(* Logix 5000 project; controller LeakTestAuto vendor 1 type 14 code 226 rev 37.11; software revision 37.01 *)

TASK MainTask (continuous, watchdog 500 ms) : MainProgram
TASK SafetyTask (periodic, rate 20 ms, priority 10, watchdog 20 ms, safety) : SafetyProgram

MODULES
   Local : vendor 1 type 14 code 226 (5069 0, rev 37.11)
      Main : vendor 1 type 14 code 195 (Ethernet 192.168.1.210, rev 33.1, $87205a54$ RPI 20 ms)
       : 5069-IB8S (5069 1, rev 2.1, SafetyInput RPI 20 ms)
      Barcode : vendor 367 type 43 code 1009 (Ethernet 192.168.1.214, rev 1.1, StandardDataDriven RPI 20 ms)
      CTS1 : vendor 1415 type 43 code 9245 (Ethernet 192.168.1.212, rev 1.1, StandardDataDriven RPI 25 ms)
      CTS2 : vendor 1415 type 43 code 9245 (Ethernet 192.168.1.213, rev 1.1, StandardDataDriven RPI 25 ms)
      EpsonRobot : vendor 1009 type 43 code 9 (Ethernet 192.168.1.215, rev 1.2, StandardDataDriven RPI 10 ms)
       : 5069-IB16 (5069 3, rev 2.1, StandardDataDriven RPI 5 ms)
       : 5069-OB16 (5069 5, rev 3.1, StandardDataDriven RPI 5 ms)
       : 5069-IB16 (5069 4, rev 2.1, StandardDataDriven RPI 5 ms)
       : 5069-OBV8S (5069 2, rev 1.1, SafetyInput RPI 20 ms)
      RFID : vendor 322 type 43 code 102 (Ethernet 192.168.1.217, rev 4.2, StandardDataDriven RPI 10 ms)
      DTE102_RFID_LoadingNest : vendor 322 type 43 code 102 (Ethernet 192.168.1.218, rev 4.2, StandardDataDriven RPI 10 ms)
END_MODULES

TYPE DTE102_CmdModule :   // It handles the imapping of the DTE102 command and status
STRUCT
   ActivateCommand : DTE102_OutputBits;   // Used to give commmands to DTE102 from PLC
   Status : DTE102_InputBits;   // Used to read the status from the DTE102 to PLC
END_STRUCT
END_TYPE

TYPE DTE102_InputBits :   // List of Bits used in PLC Input Image
STRUCT
   TP : BOOL;   // Byte 1, Bit 0 - Tag Present Status
   AI : BOOL;   // Byte 1, Bit 1 - Antenna Inactive Status
   WA : BOOL;   // Byte 1, bit 2 - Mode Write Data ACTIVE
   RA : BOOL;   // Byte 1, bit 3 - Mode Read Data ACTIVE
   UA : BOOL;   // Byte 1, bit 4 - Mode User Data Access ACTIVE
   EA : BOOL;   // Byte 1, bit 5 - Mode Receive User Data on Event Change ACTIVE
   DA : BOOL;   // Byte 1, bit 6 - Mode Diagnostics Read ACTIVE
   DIAG : BOOL;   // Byte 1, bit 7 - DIAGnostic Data Present
   TA : BOOL;   // Byte 2, bit 0 - Toggle Request Acknowledge
   CA : BOOL;   // Byte 2, bit 7 - Command Mode Active
END_STRUCT
END_TYPE

TYPE DTE102_OutputBits :   // List of Bits used in PLC Output Image
STRUCT
   AO : BOOL;   // Byte 1, Bit 1 - Antenna Inactive Request
   WR : BOOL;   // Byte 1, bit 2 - Mode Write Data ACTIVATE Command
   RD : BOOL;   // Byte 1, bit 3 - Mode Read Data ACTIVATE Command
   UR : BOOL;   // Byte 1, bit 4 - Mode User Data Access ACTIVATE Command
   ER : BOOL;   // Byte 1, bit 5 - Event Controlled reading of user memory of the ID tag
   DR : BOOL;   // Byte 1, bit 6 - Mode Diagnostics Read
   TR : BOOL;   // Byte 2, bit 0 - Toggle Request
   CM : BOOL;   // Byte 2, bit 7 - Command Mode Activate
END_STRUCT
END_TYPE

TYPE STR_Barcode :
STRUCT
   LEN : DINT;
   DATA : SINT[128];
END_STRUCT
END_TYPE

TYPE STRING16 :
STRUCT
   LEN : DINT;
   DATA : SINT[16];
END_STRUCT
END_TYPE

TYPE String20 :
STRUCT
   LEN : DINT;
   DATA : SINT[20];
END_STRUCT
END_TYPE

TYPE String35 :
STRUCT
   LEN : DINT;
   DATA : SINT[35];
END_STRUCT
END_TYPE

TYPE STRING80 :
STRUCT
   LEN : DINT;
   DATA : SINT[80];
END_STRUCT
END_TYPE

TYPE udt_CTS_INPUTS_FROM :
STRUCT
   Discrete_Status_Data : INT;   // Discrete Type Instrument Outputs
   Discrete_User_Output : INT;   // Control Commands
   Active_program_num : INT;   // Current program number
   Active_child_program : INT;   // required for alignment
   unique_id : DINT;   // Unique Identifier for the most recent result
   channel_num : SINT;   // Channel number for the most recent result
   Reserved_4 : SINT;
   Reserved_5 : SINT;
   Reserved_6 : SINT;
   program_num : INT;   // Program number for the most recent result
   sequence_num : INT;   // Test Port number for the most recent result
   seq_unique_ID : DINT;   // UID of seq program
   evaluation_code : INT;   // Evaluation code for the most recent result
   test_port : SINT;   // Test Port
   year : SINT;   // Timestamp year (YY) for the most recent result
   month : SINT;   // Timestamp month (MM) for the most recent result
   date : SINT;   // Timestamp day (DD) for the most recent result
   hour : SINT;   // Timestamp hour (HH) for the most recent result
   minutes : SINT;   // Timestamp minute (MM) for the most recent result
   seconds : SINT;   // Timestamp second (SS) for the most recent result
   flags : SINT;   // Result flags
   test_type : INT;   // Test Type
   Segment_code : INT;
   Measurement_data : udt_CTS_Measurement_Element[4];
END_STRUCT
END_TYPE

TYPE udt_CTS_Measurement_Element :
STRUCT
   Variable_code : INT;
   Variable_Number : SINT;
   Precision_code : SINT;
   Unit_code : INT;
   Reserved_1 : SINT;
   Reserved_2 : SINT;
   result_measurement : REAL;
END_STRUCT
END_TYPE

TYPE udt_CTS_OUTPUTS_TO :
STRUCT
   reserved : BOOL;   // reserved1
   change_program : BOOL;   // out_value 1
   Latch_2_Clear : BOOL;   // out_value 2
   Latch_2_Set : BOOL;   // out_value 3
   Latch_1_Clear : BOOL;   // out_value 4
   Latch_1_Set : BOOL;   // out_value 5
   New_Result_Clear : BOOL;   // out_value 6
   Requested_Result_Clear : BOOL;   // out_value 7
   reserved_2 : BOOL;   // out_value 8
   reserved_3 : BOOL;   // out_value 9
   reerved_4 : BOOL;   // out_value 10
   reserved_5 : BOOL;   // out_value 11
   vent_halt : BOOL;   // out_value 12
   reset : BOOL;   // out_value 13
   Stop : BOOL;   // out_value 14
   Start_channel : BOOL;   // out_value 15
   Out_val_1 : BOOL;   // out_value 16
   Out_val_2 : BOOL;   // Change_Program
   Out_val_3 : BOOL;   // Latch_2_Clear
   Out_val_4 : BOOL;   // Latch_2_Set
   Out_val_5 : BOOL;   // Latch_1_Clear
   Out_val_6 : BOOL;   // Latch_1_Set
   Out_val_7 : BOOL;   // New Result Clear
   Out_val_8 : BOOL;   // Requested Result Clear
   Out_val_9 : BOOL;   // reserved3
   Out_val_10 : BOOL;   // reserved4
   Out_val_11 : BOOL;   // reserved5
   Out_val_12 : BOOL;   // reserved6
   Out_val_13 : BOOL;   // VentHalt
   Out_val_14 : BOOL;   // Reset
   Out_val_15 : BOOL;   // Stop
   Out_val_16 : BOOL;   // Start_Channel
   program_num : INT;   // program_num
END_STRUCT
END_TYPE

TYPE udt_CTS_RESULT :
STRUCT
   UID : DINT;
   Basic : udt_CTS_RESULT_BASIC;
   Detailed : udt_CTS_RESULT_DETAILED;
END_STRUCT
END_TYPE

TYPE udt_CTS_RESULT_BASIC :
STRUCT
   unique_id : DINT;
   channel_num : SINT;
   reserved1 : SINT;
   reserved2 : SINT;
   reserved3 : SINT;
   program_num : INT;
   sequence_num : SINT;
   seq_unique_ID : DINT;
   evaluation_code : INT;
   test_port : SINT;
   year : SINT;
   month : SINT;
   date : SINT;
   hour : SINT;
   minute : SINT;
   second : SINT;
   reserved_4 : SINT;
   flags : SINT;
   reserved_5 : SINT;
   barcode_characters : SINT[80];
   Num_tests : SINT;
   reserved_6 : SINT;
   reserved_7 : SINT;
   reserved_8 : SINT;
   test_elements : udt_CTS_RESULT_BASIC_TEST_ELEMENT;
   barcode : STRING80;
END_STRUCT
END_TYPE

TYPE udt_CTS_RESULT_BASIC_TEST_ELEMENT :
STRUCT
   test_type : INT;
   test_eval : INT;
   num_elements : SINT;
   reserved1 : SINT;
END_STRUCT
END_TYPE

TYPE udt_CTS_RESULT_DETAILED :
STRUCT
   unique_id : DINT;
   num_elements : SINT;
   reserved_1 : SINT;
   Test_Type : INT;
   element_data : udt_CTS_RESULT_DETAILED_DATA_ELEMENT[30];
   reserved_2 : SINT;
   reserved_3 : SINT;
END_STRUCT
END_TYPE

TYPE udt_CTS_RESULT_DETAILED_DATA_ELEMENT :
STRUCT
   Variable_code : INT;
   variable_Num : SINT;
   prec_code : SINT;
   Unit_code : INT;
   reserved1 : SINT;
   reserved2 : SINT;
   result_measurement : REAL;
END_STRUCT
END_TYPE

TYPE udt_DUTHistory :
STRUCT
   Barcode : STR_Barcode;
   VolumeTest : REAL;
   LeakTest : REAL;
END_STRUCT
END_TYPE

TYPE udt_EIPTemplateData :
STRUCT
   Data : SINT[64];
END_STRUCT
END_TYPE

TYPE udt_EIPTemplateLocalInput :
STRUCT
   Ready : BOOL;
   Error : BOOL;
   Busy : BOOL;
   DataAvailable : BOOL;
   Complete : BOOL;
   Spare5 : BOOL;
   Spare6 : BOOL;
   Spare7 : BOOL;
   Data : SINT[8];
   SpareB9_63 : SINT[55];
END_STRUCT
END_TYPE

TYPE udt_EIPTemplateLocalOutput :
STRUCT
   Start : BOOL;
   Stop : BOOL;
   GetData : BOOL;
   Spare3 : BOOL;
   Spare4 : BOOL;
   Spare5 : BOOL;
   Spare6 : BOOL;
   Spare7 : BOOL;
   SpareB1_63 : SINT[63];
END_STRUCT
END_TYPE

TYPE udt_EpsonInputs :
STRUCT
   ib_Initializing : BOOL;
   ib_Ready : BOOL;
   ib_Running : BOOL;
   ib_Paused : BOOL;
   ib_Error : BOOL;
   ib_EStop : BOOL;
   ib_MotorsOn : BOOL;
   ib_IsHome : BOOL;
   ib_InPos : BOOL;
   ib_GripOpen : BOOL;
   ib_GripClosed : BOOL;
   SPAREB13 : BOOL;
   SPAREB14 : BOOL;
   SPAREB15 : BOOL;
   SPAREB16 : BOOL;
   SPAREB17 : BOOL;
   iB_SpeedEcho : USINT;
   SPAREB307 : USINT;
   iB_AccEcho : USINT;
   iB_DecEcho : USINT;
   SPAREW4 : UINT;
   SPAREW5 : UINT;
   SPAREW6 : UINT;
   SPAREW7 : UINT;
   iW_PositionEcho : UINT;
   iR_X : REAL;
   iR_Y : REAL;
   iR_Z : REAL;
   iR_U : REAL;
END_STRUCT
END_TYPE

TYPE udt_EpsonOutputs :
STRUCT
   ob_Start : BOOL;
   ob_StopNOTUSED : BOOL;
   ob_Resume : BOOL;
   ob_Pause : BOOL;
   ob_Reset : BOOL;
   ob_GoHome : BOOL;
   SPAREB06 : BOOL;
   SPAREB07 : BOOL;
   ob_SpeedOverride : BOOL;
   ob_AccOverride : BOOL;
   ob_CoordMode : BOOL;
   SPAREB13 : BOOL;
   SPAREB14 : BOOL;
   SPAREB15 : BOOL;
   SPAREB16 : BOOL;
   SPAREB17 : BOOL;
   oB_SpeedPerc : USINT;
   SPAREB307 : USINT;
   oB_AccPerc : USINT;
   oB_DecPerc : USINT;
   SPAREW4 : UINT;
   SPAREW5 : UINT;
   SPAREW6 : UINT;
   SPAREW7 : UINT;
   oW_TargetPosition : UINT;
   oR_X : REAL;
   oR_Y : REAL;
   oR_Z : REAL;
   oR_U : REAL;
END_STRUCT
END_TYPE

TYPE udt_KeyenceScannerInputs :
STRUCT
   Error : BOOL;
   ResultDataAvailable : BOOL;
   ResultDataStrobe : BOOL;
   Reserve0_3 : BOOL;
   Reserve0_4 : BOOL;
   Reserve0_5 : BOOL;
   BufferOverflowError : BOOL;
   GeneralError : BOOL;
   BUSY : BOOL;
   TRGBUSY : BOOL;
   LOCKBUSY : BOOL;
   MODEBUSY : BOOL;
   ERRBUSY : BOOL;
   Reserve0_13 : BOOL;
   READY : BOOL;
   Reserve0_15 : BOOL;
   ReadComplete : BOOL;
   PresetComplete : BOOL;
   RegisterPresetDataComplete : BOOL;
   TuneComplete : BOOL;
   BloadComplete : BOOL;
   Reserve2_5 : BOOL;
   Reserve2_6 : BOOL;
   EXTRequestComplete : BOOL;
   ReadFailure : BOOL;
   PresetFailure : BOOL;
   RegisterPresetDataFailure : BOOL;
   TuneFailure : BOOL;
   BloadFailure : BOOL;
   Reserve2_13 : BOOL;
   Reserve2_14 : BOOL;
   EXTRequestFailure : BOOL;
   IN1Status : BOOL;
   IN2Status : BOOL;
   Reserve4_2 : BOOL;
   Reserve4_3 : BOOL;
   OUT1Status : BOOL;
   OUT2Status : BOOL;
   OUT3Status : BOOL;
   Reserve4_7 : BOOL;
   Unstable : BOOL;
   MatchingLevelUnstable : BOOL;
   ISOIEC15415Unstable : BOOL;
   AIMDPMUnstable : BOOL;
   SAEAS9132Unstable : BOOL;
   ISOIEC15416Unstable : BOOL;
   Reserve4_14 : BOOL;
   Reserve4_15 : BOOL;
   Reserve6_0 : BOOL;
   Reserve6_1 : BOOL;
   Reserve6_2 : BOOL;
   Reserve6_3 : BOOL;
   Reserve6_4 : BOOL;
   Reserve6_5 : BOOL;
   Reserve6_6 : BOOL;
   Reserve6_7 : BOOL;
   Reserve6_8 : BOOL;
   Reserve6_9 : BOOL;
   Reserve6_10 : BOOL;
   Reserve6_11 : BOOL;
   Reserve6_12 : BOOL;
   Reserve6_13 : BOOL;
   MatchingLevel : UINT;
   ISOIEC15415Grade : UINT;
   AIMDPMGrade : UINT;
   ISOIEC15416Grade : UINT;
   ReadResultCode : UINT;
   PresetResultCode : UINT;
   RegisterPresetDataResultCode : UINT;
   TuneResultCode : UINT;
   BloadResultCode : UINT;
   Reserve26_0 : UINT;
   Reserve28_0 : UINT;
   EXTRequestResultCode : UINT;
   GeneralErrorCode : UINT;
   SlaveID : UINT;
   ResultDataReadyCount : UINT;
   ResultDataUpdateCount : UINT;
   MasterTriggerCount : UINT;
   ResultDataSize : INT;
   ResultData : SINT[128];
END_STRUCT
END_TYPE

TYPE udt_KeyenceScannerOutputs :
STRUCT
   Reserve0_0 : BOOL;
   ResultDataLatch : BOOL;
   Reserve0_2 : BOOL;
   Reserve0_3 : BOOL;
   Reserve0_4 : BOOL;
   Reserve0_5 : BOOL;
   Reserve0_6 : BOOL;
   ErrorClear : BOOL;
   ReadRequest : BOOL;
   PresetRequest : BOOL;
   RegisterPresetDataRequest : BOOL;
   TuneRequest : BOOL;
   BloadRequest : BOOL;
   Reserve0_13 : BOOL;
   Reserve0_14 : BOOL;
   Reserve0_15 : BOOL;
   ReadCompleteClear : BOOL;
   PresetCompleteClear : BOOL;
   RegisterPresetDataCompleteClear : BOOL;
   TuneCompleteClear : BOOL;
   BloadCompleteClear : BOOL;
   Reserve2_5 : BOOL;
   Reserve2_6 : BOOL;
   EXTRequestCompleteClear : BOOL;
   Reserve2_8 : BOOL;
   Reserve2_9 : BOOL;
   Reserve2_10 : BOOL;
   Reserve2_11 : BOOL;
   Reserve2_12 : BOOL;
   Reserve2_13 : BOOL;
   Reserve2_14 : BOOL;
   Reserve2_15 : BOOL;
   BankNumber : UINT;
   Reserve6_0 : UINT;
   Reserve8_0 : UINT;
   UserDataSize : UINT;
   UserData : USINT[64];
END_STRUCT
END_TYPE

TYPE udt_Mode :
STRUCT
   PowerOn : BOOL;
   PowerOnONS : BOOL;
   PowerOnPulse : BOOL;
   AirOk : BOOL;
   UtilitiesOk : BOOL;
   EStopsOk : BOOL;
   GuardDoorsOk : BOOL;
   FaultActive : BOOL;
   WarningActive : BOOL;
   MessageActive : BOOL;
   AutoMode : BOOL;
   ReadyForAuto : BOOL;
   ManualMode : BOOL;
   StepMode : BOOL;
   AutoMode_PB : BOOL;
   ManualMode_PB : BOOL;
   FaultReset_PB : BOOL;
   ClearFaults : BOOL;
   StepMode_PB : BOOL;
   StepMode_ONS : BOOL;
   StepMode_IND : BOOL;
   StepModeToggle : BOOL;
   Homing : BOOL;
   Home : BOOL;
   HomingCycleOvertime : BOOL;
   HomeStation_PB : BOOL;
   UpdateFaultStep : BOOL;
   InCycle : BOOL;
   CycleStart_PB : BOOL;
   CycleStop_PB : BOOL;
   CyclePause_PB : BOOL;
   CycleStopOveride : BOOL;
   CycleStopRequested : BOOL;
   CyclePauseRequested : BOOL;
   SequenceEnable : BOOL;
   DryCycle : BOOL;
   DryCycle_PB : BOOL;
   DryCycle_IND : BOOL;
   DryCycle_ONS : BOOL;
   LampTest : BOOL;
   LampTest_PB : BOOL;
   LampTest_IND : BOOL;
   LampTest_ONS : BOOL;
   Purge : BOOL;
   Purge_PB : BOOL;
   Purge_IND : BOOL;
   Purge_ONS : BOOL;
   MESBypass : BOOL;
   MESBypass_PB : BOOL;
   MESBypass_IND : BOOL;
   MESBypass_ONS : BOOL;
   StationIsEmpty : BOOL;
   ManualMode_IND : SINT;
   Home_IND : SINT;
   AutoMode_IND : SINT;
   InCycle_IND : SINT;
   CycleStop_IND : SINT;
   CyclePause_IND : SINT;
   HMIBackgroundIND : DINT;
   AlarmBannerIND : DINT;
   Faults : DINT[2];
   Warnings : DINT[1];
   Messages : DINT[3];
   HomingOvertime : TIMER;
   PowerOnTMR : TIMER;
   AirOKTMR : TIMER;
   CycleStopOverideTMR : TIMER;
   FaultTMR : udt_Timer32[2];
   WarningTMR : udt_Timer32[1];
END_STRUCT
END_TYPE

TYPE udt_OutputStructure :
STRUCT
   IL : BOOL;   // Interlock
   PB : BOOL;   // Pushbutton
   CMD : BOOL;   // Command
   BC : BOOL;   // Backcheck
   Faulted : BOOL;
   IND : SINT;   // Indicator 0 = Gray = No IL 1 = Blue = IL 2 = Green = Home 3 = Yellow = Work 4 = Red = Faulted
   REQ : SINT;   // Request
   Step : INT[8];
   FaultStep : INT[1];
   BTMR : TIMER;   // Backcheck Timer
END_STRUCT
END_TYPE

TYPE udt_ProcessFault :
STRUCT
   RowFault : BOOL;   // 3 In A Row Fault
   HourFault : BOOL;   // 5 In A Hour Fault
   ShiftFault : BOOL;   // 10 In A Shift Fault
   RowCount : DINT;
   HourCount : DINT;
   ShiftCount : DINT;
   RowPalletHist : DINT[3];
   RowPalletHistBuffer : DINT[3];
   HourPalletHist : DINT[5];
   HourPalletHistBuffer : DINT[5];
   ShiftPalletHist : DINT[10];
   ShiftPalletHistBuffer : DINT[10];
END_STRUCT
END_TYPE

TYPE udt_Produced_SetTime :
STRUCT
   SetTimePB : BOOL;
   SetTime : DINT[6];
END_STRUCT
END_TYPE

TYPE udt_SequenceStructure_X64 :
STRUCT
   SequenceRunning : BOOL;
   WorkReqd : BOOL;
   NoWorkReqd : BOOL;
   ProcessComplete : BOOL;
   CycleDone : BOOL;
   ResetMemories : BOOL;
   NextStepPB : BOOL;
   CalculateStepTime : BOOL;
   CurrentStep : INT;
   NextStep : INT;
   StepTimePointer : INT;
   ONS : INT;
   StepHistory : INT[64];
   StepHistoryPointer : INT;
   StepDescriptionPointer : INT;
   CurrentCycleTime : REAL;
   AverageCycleTime : REAL;
   PreviousCycleTime : REAL;
   CycleTimeHistory : REAL[10];
   CurrentStepCycleTime : REAL;
   StepTimeHistory : REAL[64];
   NominalStepTimeHistory : REAL[64];
   StepTimer : TIMER;
   CycleTimer : TIMER;
   CycleDoneDelayTMR : TIMER;
   HMI_CurrentStepDescription : String35;
   StepDescriptions : String35[64];
END_STRUCT
END_TYPE

TYPE udt_Timer32 :
STRUCT
   TMR : TIMER[32];
END_STRUCT
END_TYPE

ADD_ON_INSTRUCTION AOI_CommStatus   (* revision 1.0 *)
VAR_IN_OUT
   Module : MODULE; {required}
END_VAR
VAR_INPUT
   Cmd : BOOL; {required}
END_VAR
VAR_OUTPUT
   stsStandby : BOOL; {access Read Only, visible}
   stsFaulted : BOOL; {access Read Only, visible}
   stsValidating : BOOL; {access Read Only, visible}
   stsConnecting : BOOL; {access Read Only, visible}
   stsRunning : BOOL; {access Read Only, visible}
   stsShuttingDown : BOOL; {access Read Only, visible}
   stsInhibited : BOOL; {access Read Only, visible}
   stsWaiting : BOOL; {access Read Only, visible}
   stsFirmwareUpdating : BOOL; {access Read Only, visible}
   stsConfiguring : BOOL; {access Read Only, visible}
   stsFaultCode : DINT; {access Read Only, visible}
END_VAR
VAR
   Status : DINT; {access None}
   ons : BOOL; {access None}
   CmdOns : BOOL; {access None}
END_VAR

ROUTINE Logic   (* ladder *)
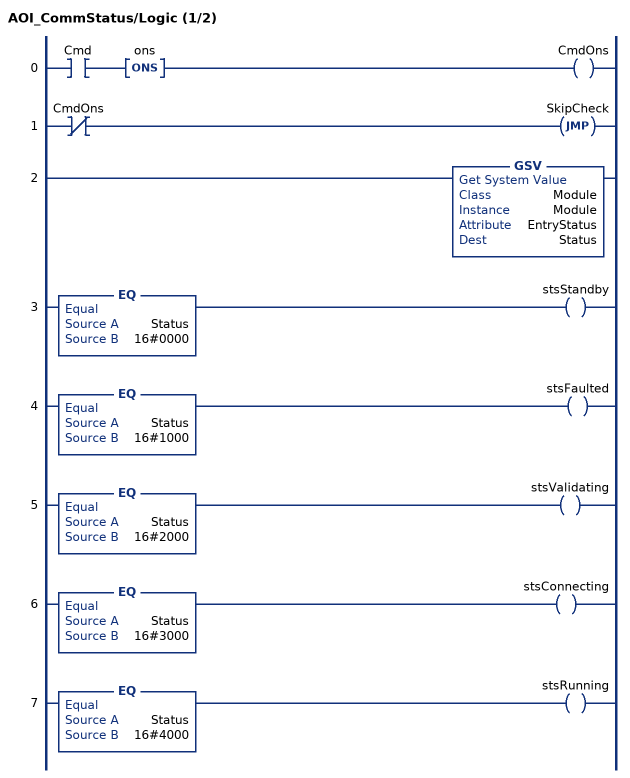
   0: XIC(Cmd)ONS(ons)OTE(CmdOns);
   1: XIO(CmdOns)JMP(SkipCheck);
   2: GSV(Module,Module,EntryStatus,Status);
   3: EQ(Status,16#0000)OTE(stsStandby);
   4: EQ(Status,16#1000)OTE(stsFaulted);
   5: EQ(Status,16#2000)OTE(stsValidating);
   6: EQ(Status,16#3000)OTE(stsConnecting);
   7: EQ(Status,16#4000)OTE(stsRunning);
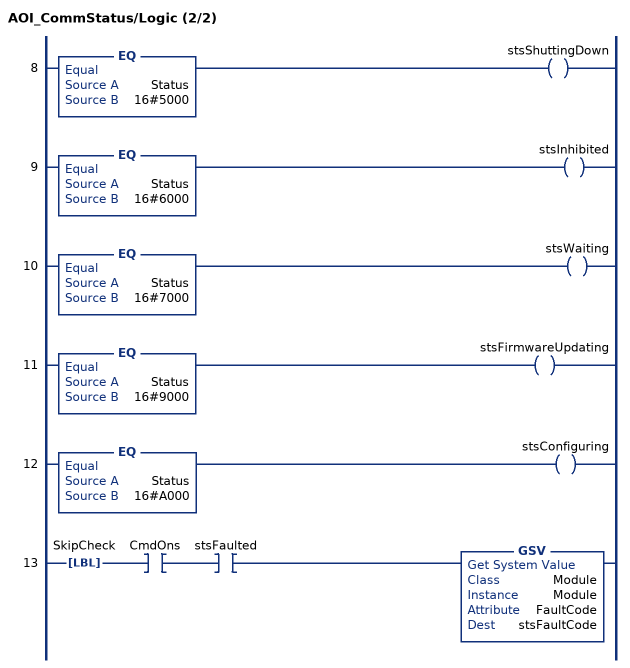
   8: EQ(Status,16#5000)OTE(stsShuttingDown);
   9: EQ(Status,16#6000)OTE(stsInhibited);
   10: EQ(Status,16#7000)OTE(stsWaiting);
   11: EQ(Status,16#9000)OTE(stsFirmwareUpdating);
   12: EQ(Status,16#A000)OTE(stsConfiguring);
   13: LBL(SkipCheck)XIC(CmdOns)XIC(stsFaulted)GSV(Module,Module,FaultCode,stsFaultCode);
END_ROUTINE
END_ADD_ON_INSTRUCTION

ADD_ON_INSTRUCTION AOI_CTS_INSTRUMENT   (* revision 2.0, vendor Cincinnati Test Systems *)
// Revision note:
// Rev 2.0 for rectifed eds and corrected tags
VAR_IN_OUT
   Input : udt_CTS_INPUTS_FROM; {required}
   Output : udt_CTS_OUTPUTS_TO; {required}
END_VAR
VAR_INPUT
   Write_Barcode_Trigger : BOOL; {visible}
END_VAR
VAR_OUTPUT
   Write_Barcode_Complete : BOOL; {access Read Only, visible}
END_VAR
VAR_INPUT
   Read_Barcode_Trigger : BOOL; {visible}
END_VAR
VAR_OUTPUT
   Read_Barcode_Complete : BOOL; {access Read Only, visible}
END_VAR
VAR_IN_OUT
   Barcode_Data_To_Write : STRING80; {required}
   Barcode_Data_Read : STRING80; {required}
   Barcode_Write_Message : MESSAGE; {required}
   Barcode_Read_Message : MESSAGE; {required}
END_VAR
VAR_INPUT
   Change_Prog_Trigger : BOOL; {visible}
   Change_Program_Number : DINT; {visible}
END_VAR
VAR_OUTPUT
   Current_Program_Number : DINT; {access Read Only, visible}
END_VAR
VAR_INPUT
   Start : BOOL; {visible}
   Stop : BOOL; {visible}
   Reset : BOOL; {visible}
   Vent_Halt : BOOL; {visible}
   New_Result_Clear : BOOL; {visible}
   Latch_1_Set : BOOL;
   Latch_1_Clear : BOOL;
   Latch_2_Set : BOOL;
   Latch_2_Clear : BOOL;
   User_Input_1 : BOOL;
   User_Input_2 : BOOL;
   User_Input_3 : BOOL;
   User_Input_4 : BOOL;
   User_Input_5 : BOOL;
   User_Input_6 : BOOL;
   User_Input_7 : BOOL;
   User_Input_8 : BOOL;
   User_Input_9 : BOOL;
   User_Input_10 : BOOL;
   User_Input_11 : BOOL;
   User_Input_12 : BOOL;
   User_Input_13 : BOOL;
   User_Input_14 : BOOL;
   User_Input_15 : BOOL;
   User_Input_16 : BOOL;
END_VAR
VAR_OUTPUT
   Instrument_Ready : BOOL; {access Read Only, visible}
   Malfunction : BOOL; {access Read Only, visible}
   Program_Accept : BOOL; {access Read Only, visible}
   Program_Reject : BOOL; {access Read Only, visible}
   New_Result : BOOL; {access Read Only, visible}
   Requested_Result_Available : BOOL; {access Read Only}
   Requested_Result_Error : BOOL; {access Read Only}
   Latch_State_1 : BOOL; {access Read Only}
   Latch_State_2 : BOOL; {access Read Only}
   User_Output_1 : BOOL; {access Read Only}
   User_Output_2 : BOOL; {access Read Only}
   User_Output_3 : BOOL; {access Read Only}
   User_Output_4 : BOOL; {access Read Only}
   User_Output_5 : BOOL; {access Read Only}
   User_Output_6 : BOOL; {access Read Only}
   User_Output_7 : BOOL; {access Read Only}
   User_Output_8 : BOOL; {access Read Only}
   User_Output_9 : BOOL; {access Read Only}
   User_Output_10 : BOOL; {access Read Only}
   User_Output_11 : BOOL; {access Read Only}
   User_Output_12 : BOOL; {access Read Only}
   User_Output_13 : BOOL; {access Read Only}
   User_Output_14 : BOOL; {access Read Only}
   User_Output_15 : BOOL; {access Read Only}
   User_Output_16 : BOOL; {access Read Only}
   Last_Result_Unique_ID : DINT; {access Read Only, visible}
   Last_Result_Channel_Number : SINT; {access Read Only}
   Last_Result_Progam_Number : DINT; {access Read Only, visible}
   Last_Result_Test_Port : SINT; {access Read Only}
   Last_Result_Evaluation_Code : SINT; {access Read Only}
END_VAR
VAR_IN_OUT
   Last_Result_Evaluation : STRING16; {required}
END_VAR
VAR_OUTPUT
   Last_Result_Year : SINT; {access Read Only}
   Last_Result_Month : SINT; {access Read Only}
   Last_Result_Date : SINT; {access Read Only}
   Last_Result_Hour : SINT; {access Read Only}
   Last_Result_Minute : SINT; {access Read Only}
   Last_Result_Second : SINT; {access Read Only}
   Last_Result_Number_of_Children : SINT; {access Read Only, visible}
END_VAR
VAR_INPUT
   Get_Results_Trigger : BOOL; {visible}
END_VAR
VAR_OUTPUT
   Getting_Results : BOOL; {access Read Only}
END_VAR
VAR_INPUT
   UID_of_Desired_Results : DINT; {visible}
   Include_Detailed_Results : BOOL; {visible}
END_VAR
VAR_OUTPUT
   Results_Ready : BOOL; {access Read Only, visible}
   Results_Error : BOOL; {access Read Only}
END_VAR
VAR_IN_OUT
   Results_UID_Message : MESSAGE; {required}
   Basic_Results_Message : MESSAGE; {required}
   Detailed_Results_Message : MESSAGE; {required}
   Results : udt_CTS_RESULT; {required}
END_VAR
VAR_INPUT
   UID_Time : DINT := 1300;
END_VAR
VAR_OUTPUT
   Timeout_time : DINT; {access Read Only}
   Test_Time : DINT; {access Read Only}
   Accept_Time : DINT; {access Read Only}
   Instr_Ready : DINT; {access Read Only, required}
   Ready : BOOL; {access Read Only}
   Test_Active : BOOL; {access Read Only}
   Barcode_Flag : BOOL; {access Read Only}
   Fisrt_Scan_Allow : BOOL; {access Read Only}
END_VAR
VAR
   Get_Results_ONS : BOOL; {access None}
   Basic_Results_Conversion_Complete : BOOL; {access None}
   Detailed_Results_Conversion_Complete : BOOL; {access None}
   Error_Delay : TIMER := (PRE := 500); {access None}
   FSC_Find_Null_BC_Read : CONTROL := (LEN := 82); {access None}
   FSC_Bas_Rslt_Find_Null_BC : CONTROL := (LEN := 1); {access None}
   Last_Result_Unique_ID_Previous : DINT; {access None}
   Read_Barcode_ONS : BOOL; {access None}
   FSC_Find_Null_Last_Rslt_Eval : CONTROL; {access None}
   UID_Move : TIMER := (PRE := 300); {access None}
   Always_ON : BOOL; {access None}
   Rise_Pulse : BOOL; {access None}
   UID_send : DINT; {access None}
   UID_send_Timer : TIMER := (PRE := 4000); {access None}
   specific_UID : DINT; {access None}
   Wait_time : TIMER; {access None}
   Denied : BOOL; {access None}
   Allow : BOOL; {access None}
   Time_Elapsed : TIMER; {access None}
   Res_Ready : BOOL; {access None}
   Bypass : BOOL; {access None}
END_VAR

ROUTINE Logic   (* ladder *)
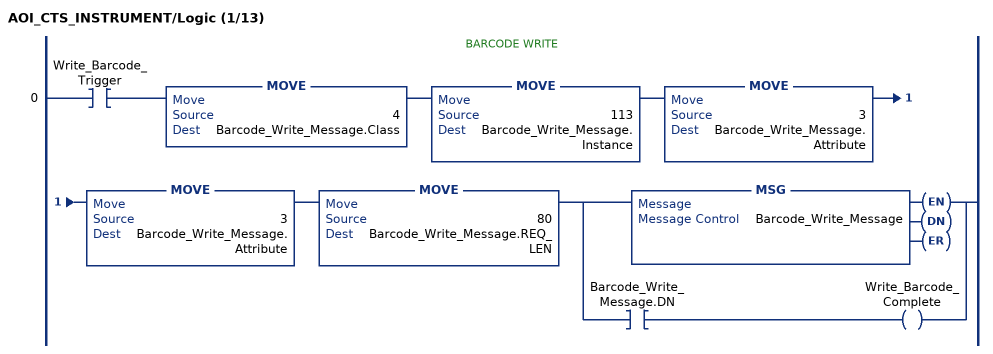
   // BARCODE WRITE
   0: XIC(Write_Barcode_Trigger)MOVE(4,Barcode_Write_Message.Class)MOVE(113,Barcode_Write_Message.Instance)MOVE(3,Barcode_Write_Message.Attribute)MOVE(3,Barcode_Write_Message.Attribute)MOVE(80,Barcode_Write_Message.REQ_LEN)[MSG(Barcode_Write_Message) ,XIC(Barcode_Write_Message.DN) OTE(Write_Barcode_Complete) ];
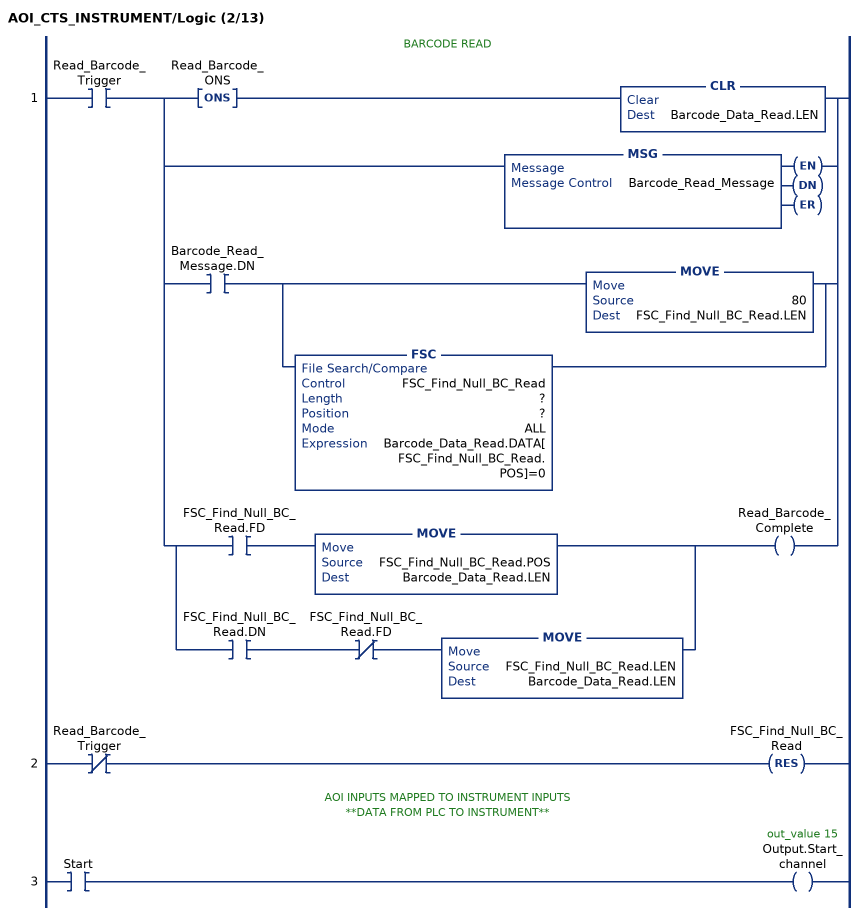
   // BARCODE READ
   1: XIC(Read_Barcode_Trigger)[ONS(Read_Barcode_ONS) CLR(Barcode_Data_Read.LEN) ,MSG(Barcode_Read_Message) ,XIC(Barcode_Read_Message.DN) [MOVE(80,FSC_Find_Null_BC_Read.LEN) ,FSC(FSC_Find_Null_BC_Read,?,?,ALL,Barcode_Data_Read.DATA[FSC_Find_Null_BC_Read.POS]=0) ] ,[XIC(FSC_Find_Null_BC_Read.FD) MOVE(FSC_Find_Null_BC_Read.POS,Barcode_Data_Read.LEN) ,XIC(FSC_Find_Null_BC_Read.DN) XIO(FSC_Find_Null_BC_Read.FD) MOVE(FSC_Find_Null_BC_Read.LEN,Barcode_Data_Read.LEN) ] OTE(Read_Barcode_Complete) ];
   2: XIO(Read_Barcode_Trigger)RES(FSC_Find_Null_BC_Read);
   // AOI INPUTS MAPPED TO INSTRUMENT INPUTS
   // **DATA FROM PLC TO INSTRUMENT**
   3: XIC(Start)OTE(Output.Start_channel);
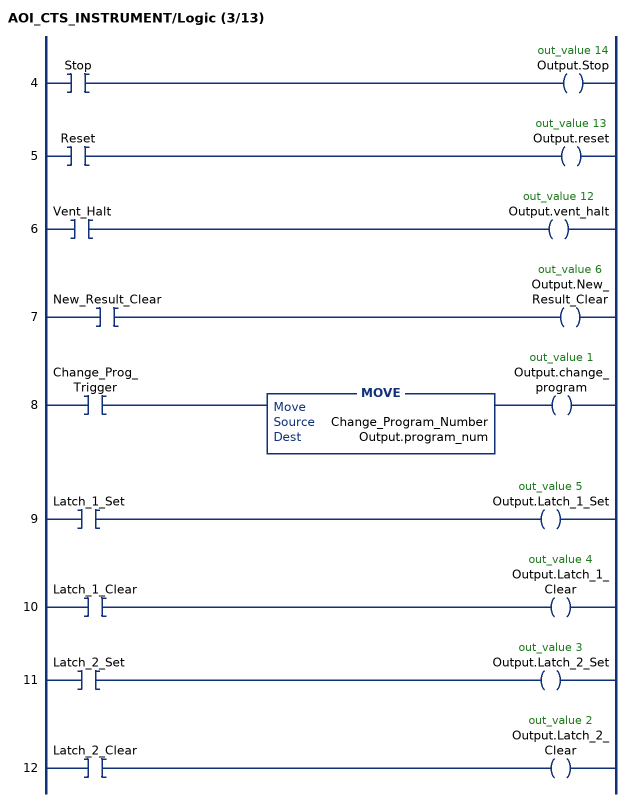
   4: XIC(Stop)OTE(Output.Stop);
   5: XIC(Reset)OTE(Output.reset);
   6: XIC(Vent_Halt)OTE(Output.vent_halt);
   7: XIC(New_Result_Clear)OTE(Output.New_Result_Clear);
   8: XIC(Change_Prog_Trigger)MOVE(Change_Program_Number,Output.program_num)OTE(Output.change_program);
   9: XIC(Latch_1_Set)OTE(Output.Latch_1_Set);
   10: XIC(Latch_1_Clear)OTE(Output.Latch_1_Clear);
   11: XIC(Latch_2_Set)OTE(Output.Latch_2_Set);
   12: XIC(Latch_2_Clear)OTE(Output.Latch_2_Clear);
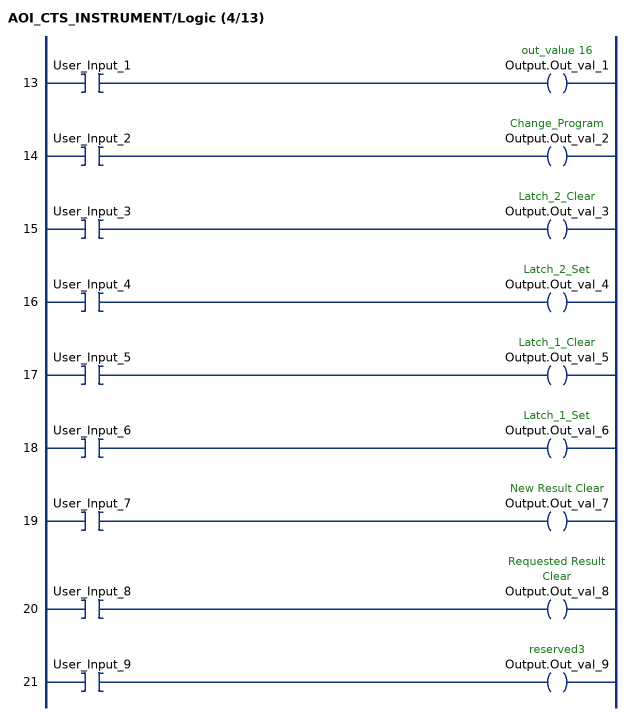
   13: XIC(User_Input_1)OTE(Output.Out_val_1);
   14: XIC(User_Input_2)OTE(Output.Out_val_2);
   15: XIC(User_Input_3)OTE(Output.Out_val_3);
   16: XIC(User_Input_4)OTE(Output.Out_val_4);
   17: XIC(User_Input_5)OTE(Output.Out_val_5);
   18: XIC(User_Input_6)OTE(Output.Out_val_6);
   19: XIC(User_Input_7)OTE(Output.Out_val_7);
   20: XIC(User_Input_8)OTE(Output.Out_val_8);
   21: XIC(User_Input_9)OTE(Output.Out_val_9);
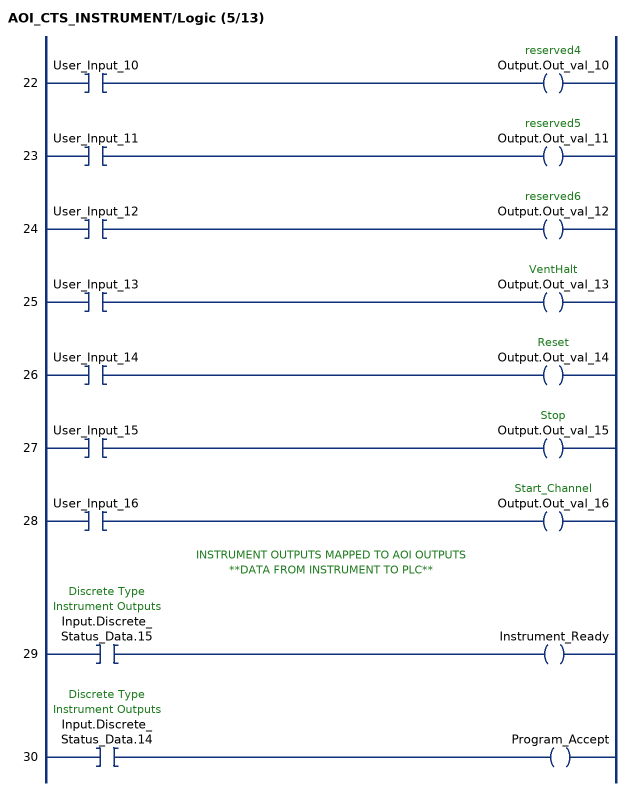
   22: XIC(User_Input_10)OTE(Output.Out_val_10);
   23: XIC(User_Input_11)OTE(Output.Out_val_11);
   24: XIC(User_Input_12)OTE(Output.Out_val_12);
   25: XIC(User_Input_13)OTE(Output.Out_val_13);
   26: XIC(User_Input_14)OTE(Output.Out_val_14);
   27: XIC(User_Input_15)OTE(Output.Out_val_15);
   28: XIC(User_Input_16)OTE(Output.Out_val_16);
   // INSTRUMENT OUTPUTS MAPPED TO AOI OUTPUTS
   // **DATA FROM INSTRUMENT TO PLC**
   29: XIC(Input.Discrete_Status_Data.15)OTE(Instrument_Ready);
   30: XIC(Input.Discrete_Status_Data.14)OTE(Program_Accept);
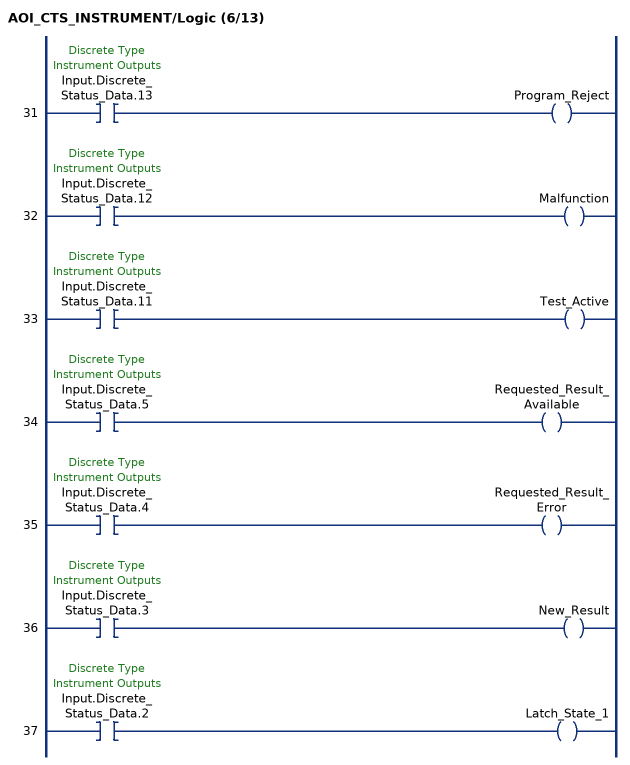
   31: XIC(Input.Discrete_Status_Data.13)OTE(Program_Reject);
   32: XIC(Input.Discrete_Status_Data.12)OTE(Malfunction);
   33: XIC(Input.Discrete_Status_Data.11)OTE(Test_Active);
   34: XIC(Input.Discrete_Status_Data.5)OTE(Requested_Result_Available);
   35: XIC(Input.Discrete_Status_Data.4)OTE(Requested_Result_Error);
   36: XIC(Input.Discrete_Status_Data.3)OTE(New_Result);
   37: XIC(Input.Discrete_Status_Data.2)OTE(Latch_State_1);
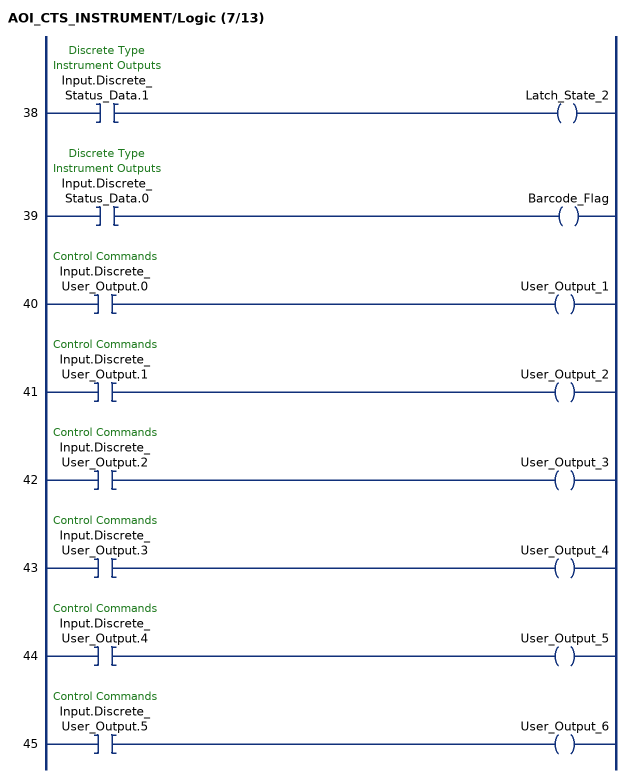
   38: XIC(Input.Discrete_Status_Data.1)OTE(Latch_State_2);
   39: XIC(Input.Discrete_Status_Data.0)OTE(Barcode_Flag);
   40: XIC(Input.Discrete_User_Output.0)OTE(User_Output_1);
   41: XIC(Input.Discrete_User_Output.1)OTE(User_Output_2);
   42: XIC(Input.Discrete_User_Output.2)OTE(User_Output_3);
   43: XIC(Input.Discrete_User_Output.3)OTE(User_Output_4);
   44: XIC(Input.Discrete_User_Output.4)OTE(User_Output_5);
   45: XIC(Input.Discrete_User_Output.5)OTE(User_Output_6);
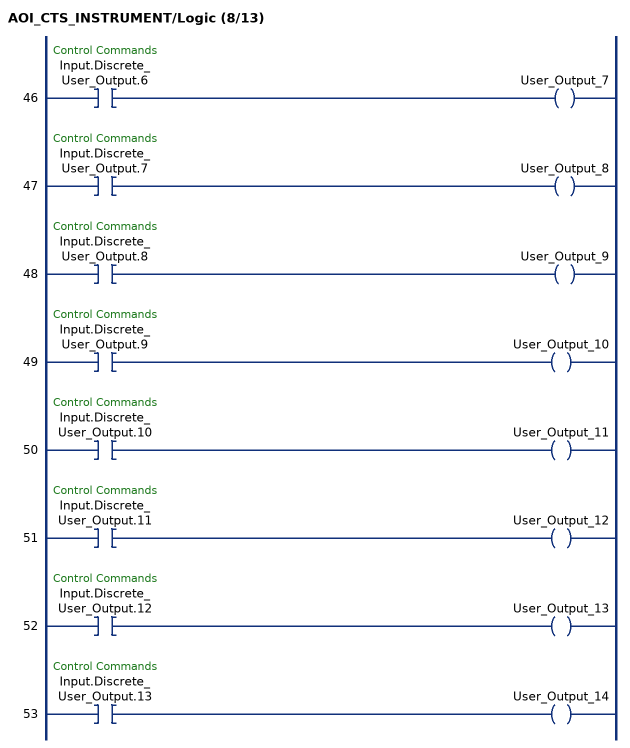
   46: XIC(Input.Discrete_User_Output.6)OTE(User_Output_7);
   47: XIC(Input.Discrete_User_Output.7)OTE(User_Output_8);
   48: XIC(Input.Discrete_User_Output.8)OTE(User_Output_9);
   49: XIC(Input.Discrete_User_Output.9)OTE(User_Output_10);
   50: XIC(Input.Discrete_User_Output.10)OTE(User_Output_11);
   51: XIC(Input.Discrete_User_Output.11)OTE(User_Output_12);
   52: XIC(Input.Discrete_User_Output.12)OTE(User_Output_13);
   53: XIC(Input.Discrete_User_Output.13)OTE(User_Output_14);
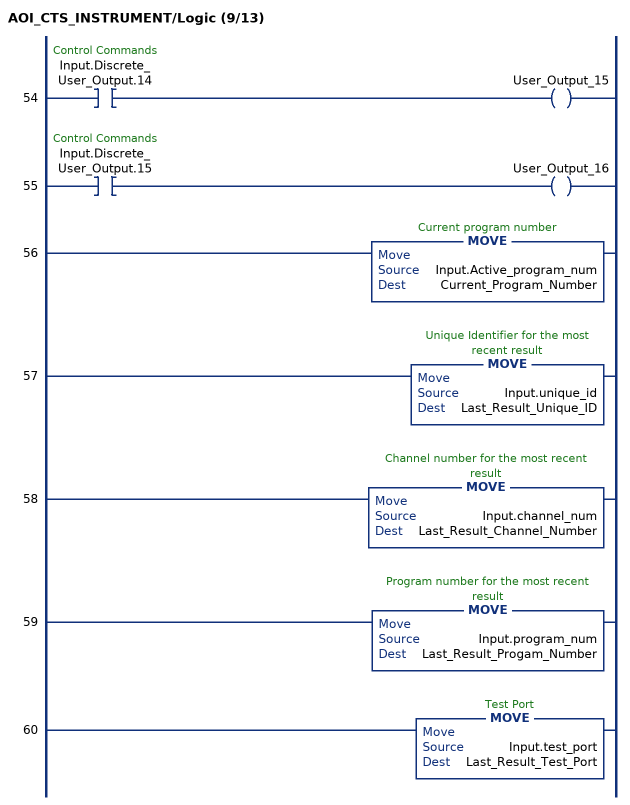
   54: XIC(Input.Discrete_User_Output.14)OTE(User_Output_15);
   55: XIC(Input.Discrete_User_Output.15)OTE(User_Output_16);
   56: MOVE(Input.Active_program_num,Current_Program_Number);
   57: MOVE(Input.unique_id,Last_Result_Unique_ID);
   58: MOVE(Input.channel_num,Last_Result_Channel_Number);
   59: MOVE(Input.program_num,Last_Result_Progam_Number);
   60: MOVE(Input.test_port,Last_Result_Test_Port);
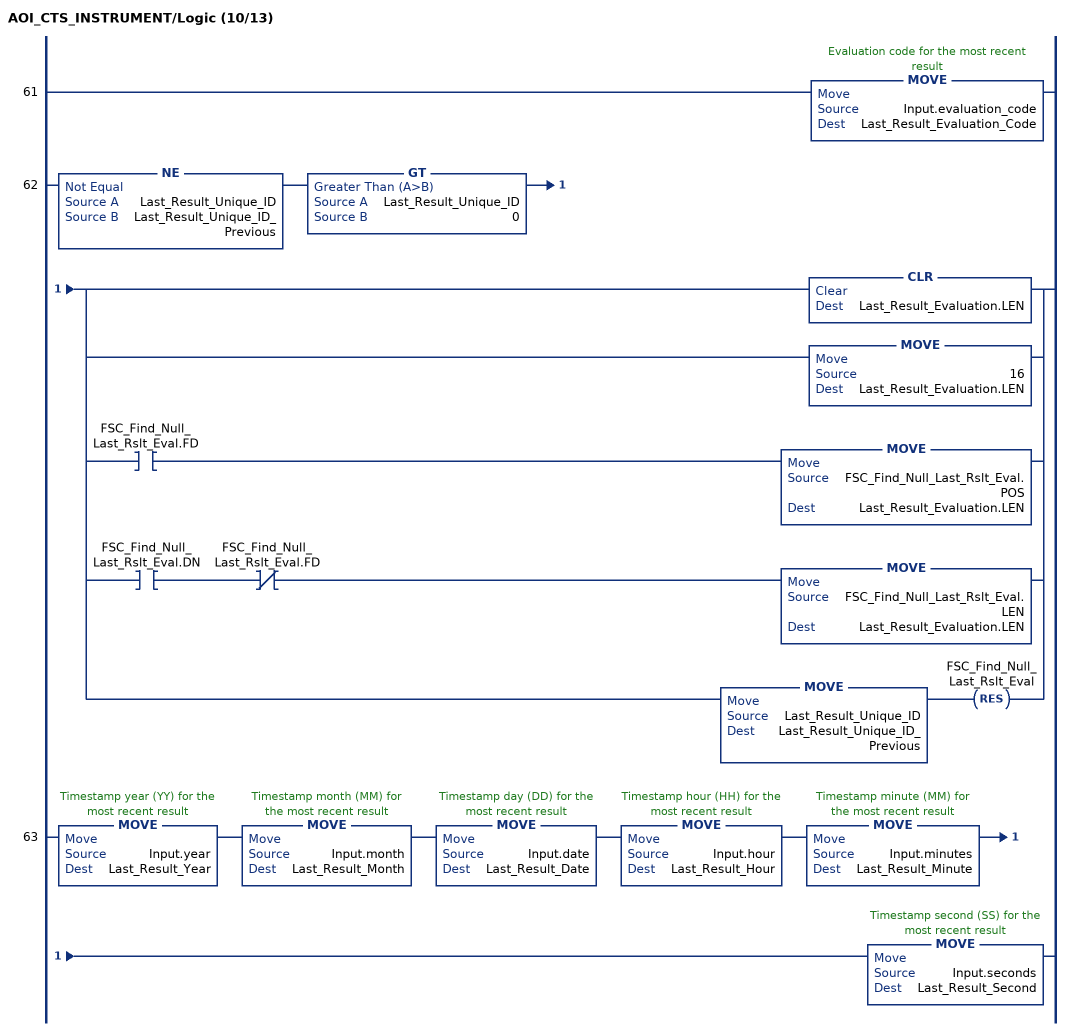
   61: MOVE(Input.evaluation_code,Last_Result_Evaluation_Code);
   62: NE(Last_Result_Unique_ID,Last_Result_Unique_ID_Previous)GT(Last_Result_Unique_ID,0)[CLR(Last_Result_Evaluation.LEN) ,MOVE(16,Last_Result_Evaluation.LEN) ,XIC(FSC_Find_Null_Last_Rslt_Eval.FD) MOVE(FSC_Find_Null_Last_Rslt_Eval.POS,Last_Result_Evaluation.LEN) ,XIC(FSC_Find_Null_Last_Rslt_Eval.DN) XIO(FSC_Find_Null_Last_Rslt_Eval.FD) MOVE(FSC_Find_Null_Last_Rslt_Eval.LEN,Last_Result_Evaluation.LEN) ,MOVE(Last_Result_Unique_ID,Last_Result_Unique_ID_Previous) RES(FSC_Find_Null_Last_Rslt_Eval) ];
   63: MOVE(Input.year,Last_Result_Year)MOVE(Input.month,Last_Result_Month)MOVE(Input.date,Last_Result_Date)MOVE(Input.hour,Last_Result_Hour)MOVE(Input.minutes,Last_Result_Minute)MOVE(Input.seconds,Last_Result_Second);
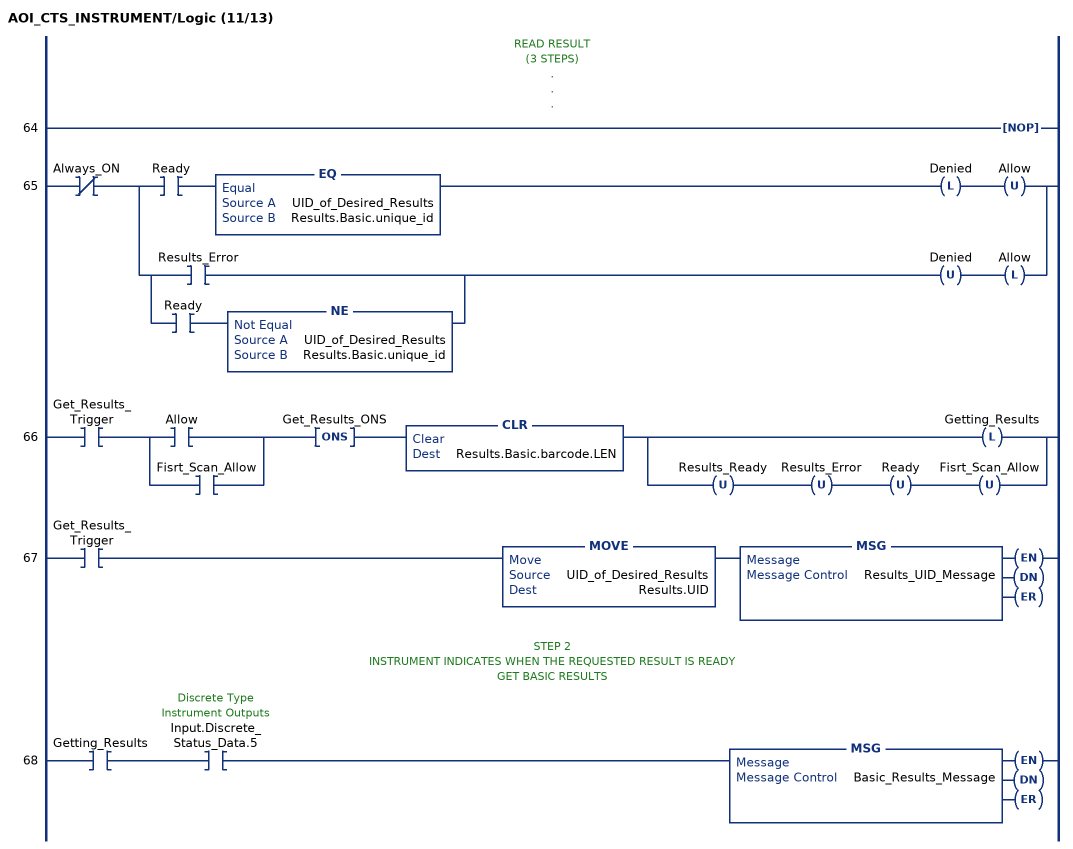
   // READ RESULT
   // (3 STEPS)
   // .
   // .
   // .
   64: NOP();
   65: XIO(Always_ON)[XIC(Ready) EQ(UID_of_Desired_Results,Results.Basic.unique_id) OTL(Denied) OTU(Allow) ,[XIC(Results_Error) ,XIC(Ready) NE(UID_of_Desired_Results,Results.Basic.unique_id) ] OTU(Denied) OTL(Allow) ];
   66: XIC(Get_Results_Trigger)[XIC(Allow) ,XIC(Fisrt_Scan_Allow) ]ONS(Get_Results_ONS)CLR(Results.Basic.barcode.LEN)[OTL(Getting_Results) ,OTU(Results_Ready) OTU(Results_Error) OTU(Ready) OTU(Fisrt_Scan_Allow) ];
   67: XIC(Get_Results_Trigger)MOVE(UID_of_Desired_Results,Results.UID)MSG(Results_UID_Message);
   // STEP 2
   // INSTRUMENT INDICATES WHEN THE REQUESTED RESULT IS READY
   // GET BASIC RESULTS
   68: XIC(Getting_Results)XIC(Input.Discrete_Status_Data.5)MSG(Basic_Results_Message);
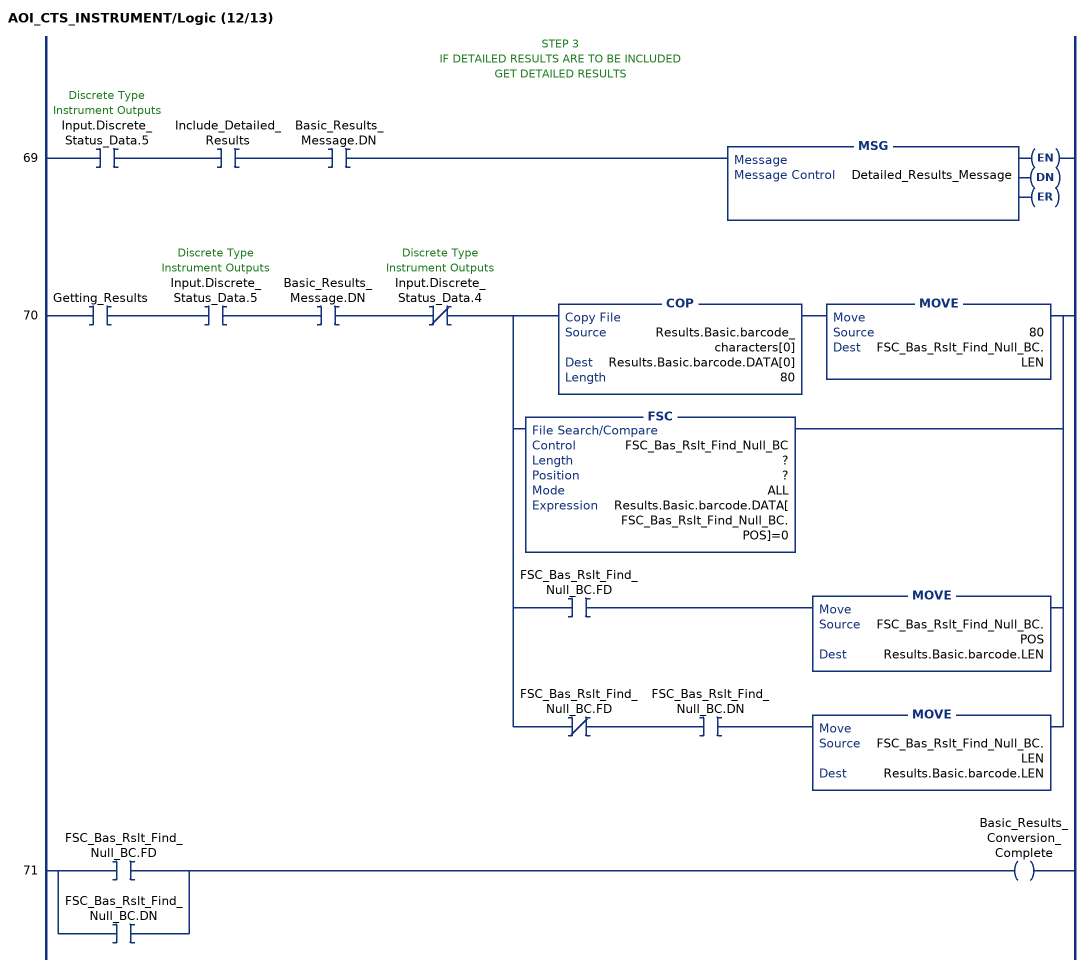
   // STEP 3
   // IF DETAILED RESULTS ARE TO BE INCLUDED
   // GET DETAILED RESULTS
   69: XIC(Input.Discrete_Status_Data.5)XIC(Include_Detailed_Results)XIC(Basic_Results_Message.DN)MSG(Detailed_Results_Message);
   70: XIC(Getting_Results)XIC(Input.Discrete_Status_Data.5)XIC(Basic_Results_Message.DN)XIO(Input.Discrete_Status_Data.4)[COP(Results.Basic.barcode_characters[0],Results.Basic.barcode.DATA[0],80) MOVE(80,FSC_Bas_Rslt_Find_Null_BC.LEN) ,[FSC(FSC_Bas_Rslt_Find_Null_BC,?,?,ALL,Results.Basic.barcode.DATA[FSC_Bas_Rslt_Find_Null_BC.POS]=0) ,[XIC(FSC_Bas_Rslt_Find_Null_BC.FD) MOVE(FSC_Bas_Rslt_Find_Null_BC.POS,Results.Basic.barcode.LEN) ,XIO(FSC_Bas_Rslt_Find_Null_BC.FD) XIC(FSC_Bas_Rslt_Find_Null_BC.DN) MOVE(FSC_Bas_Rslt_Find_Null_BC.LEN,Results.Basic.barcode.LEN) ] ] ];
   71: [XIC(FSC_Bas_Rslt_Find_Null_BC.FD) ,XIC(FSC_Bas_Rslt_Find_Null_BC.DN) ]OTE(Basic_Results_Conversion_Complete);
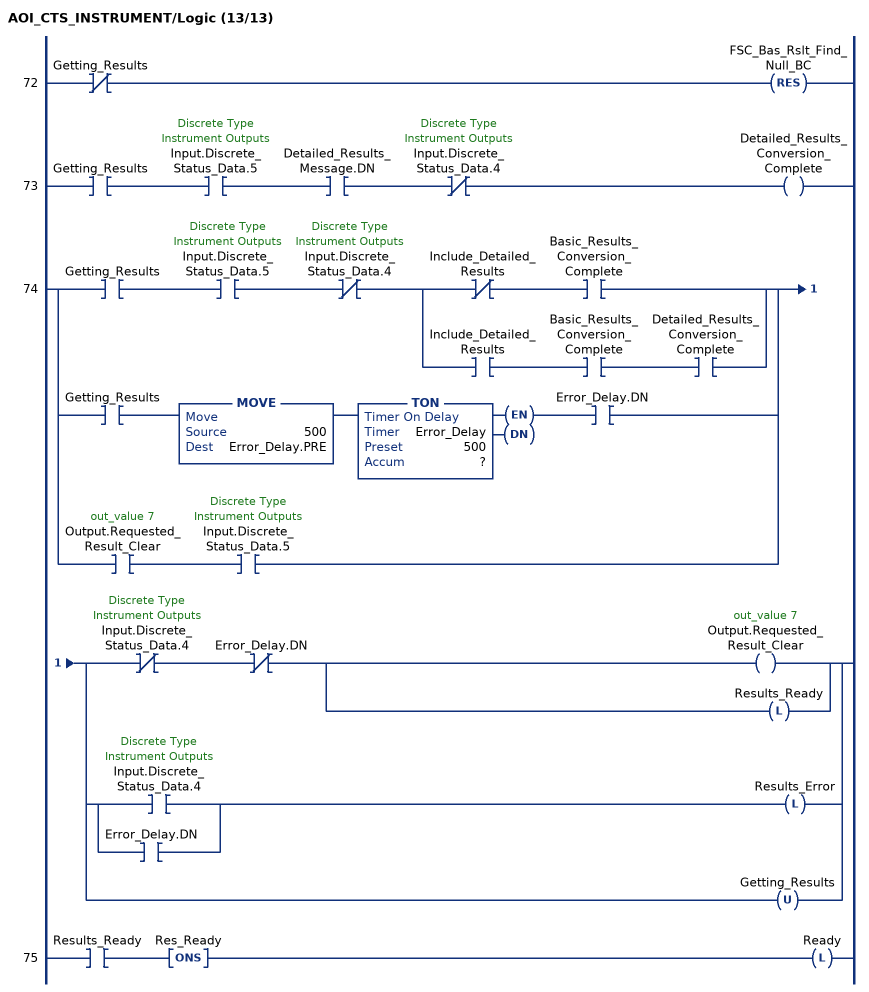
   72: XIO(Getting_Results)RES(FSC_Bas_Rslt_Find_Null_BC);
   73: XIC(Getting_Results)XIC(Input.Discrete_Status_Data.5)XIC(Detailed_Results_Message.DN)XIO(Input.Discrete_Status_Data.4)OTE(Detailed_Results_Conversion_Complete);
   74: [XIC(Getting_Results) XIC(Input.Discrete_Status_Data.5) XIO(Input.Discrete_Status_Data.4) [XIO(Include_Detailed_Results) XIC(Basic_Results_Conversion_Complete) ,XIC(Include_Detailed_Results) XIC(Basic_Results_Conversion_Complete) XIC(Detailed_Results_Conversion_Complete) ] ,XIC(Getting_Results) MOVE(500,Error_Delay.PRE) TON(Error_Delay,?,?) XIC(Error_Delay.DN) ,XIC(Output.Requested_Result_Clear) XIC(Input.Discrete_Status_Data.5) ][XIO(Input.Discrete_Status_Data.4) XIO(Error_Delay.DN) [OTE(Output.Requested_Result_Clear) ,OTL(Results_Ready) ] ,[XIC(Input.Discrete_Status_Data.4) ,XIC(Error_Delay.DN) ] OTL(Results_Error) ,OTU(Getting_Results) ];
   75: XIC(Results_Ready)ONS(Res_Ready)OTL(Ready);
END_ROUTINE
END_ADD_ON_INSTRUCTION

ADD_ON_INSTRUCTION AOI_GetShift   (* revision 1.0 *)
VAR_INPUT
   PLCHour : INT; {access Read Only, required}
END_VAR
VAR_IN_OUT
   ShiftTimes : SINT[24]; {constant, required}
END_VAR
VAR_OUTPUT
   ShiftNumber : SINT := -1; {required}
END_VAR
VAR
   numShifts : DINT; {access None}
   index : DINT; {access None}
END_VAR

ROUTINE Logic   (* structured text *)
   SIZE(ShiftTimes, 0, numShifts);
   if ShiftTimes[0]<>-1 then
   	for index := 1 to numShifts-2 do
   		if ShiftTimes[index]<>-1 then
   			if ShiftTimes[index+1]<>-1 then
   				if PLCHour>=ShiftTimes[index] AND PLCHour<ShiftTimes[index+1] then ShiftNumber := index; end_if;
   			else
   				if PLCHour>=ShiftTimes[index] OR PLCHour<ShiftTimes[0] then ShiftNumber := index; end_if;
   			end_if;
   		end_if;
   	end_for;
   	if ShiftTimes[numShifts-1] <> -1 then
   		if PLCHour>=ShiftTimes[index] OR PLCHour<ShiftTimes[0] then ShiftNumber := numShifts-1; end_if;
   	end_if;
   end_if;
END_ROUTINE
END_ADD_ON_INSTRUCTION

ADD_ON_INSTRUCTION AOI_IOCounter   (* revision 1.0 *)
VAR_IN_OUT
   ResetArray : INT[8]; {required}
   CounterArray : UDINT[128]; {required}
   HasRef : BOOL; {required}
   IOData1 : AB:5000_DI16:I:0; {required}
   IOData2 : AB:5000_DI16:I:0; {required}
   IOData3 : AB:5000_DO16:O:0; {required}
   IOData4 : AB:5000_DI16:I:0; {required}
   IOData5 : AB:5000_DI16:I:0; {required}
   IOData6 : AB:5000_DI16:I:0; {required}
   IOData7 : AB:5000_DI16:I:0; {required}
   IOData8 : AB:5000_DI16:I:0; {required}
   LastIOData : INT[8]; {required}
END_VAR
VAR
   index : DINT; {access None}
   bindex : DINT; {access None}
   CurrData : INT[8]; {access None}
END_VAR

ROUTINE Logic   (* structured text *)
   if not HasRef then
   	HasRef := 1;
   	LastIOData[0].00 := IOData1.Pt00.Data;
   	LastIOData[0].01 := IOData1.Pt01.Data;
   	LastIOData[0].02 := IOData1.Pt02.Data;
   	LastIOData[0].03 := IOData1.Pt03.Data;
   	LastIOData[0].04 := IOData1.Pt04.Data;
   	LastIOData[0].05 := IOData1.Pt05.Data;
   	LastIOData[0].06 := IOData1.Pt06.Data;
   	LastIOData[0].07 := IOData1.Pt07.Data;
   	LastIOData[0].08 := IOData1.Pt08.Data;
   	LastIOData[0].09 := IOData1.Pt09.Data;
   	LastIOData[0].10 := IOData1.Pt10.Data;
   	LastIOData[0].11 := IOData1.Pt11.Data;
   	LastIOData[0].12 := IOData1.Pt12.Data;
   	LastIOData[0].13 := IOData1.Pt13.Data;
   	LastIOData[0].14 := IOData1.Pt14.Data;
   	LastIOData[0].15 := IOData1.Pt15.Data;
   	LastIOData[1].00 := IOData2.Pt00.Data;
   	LastIOData[1].01 := IOData2.Pt01.Data;
   	LastIOData[1].02 := IOData2.Pt02.Data;
   	LastIOData[1].03 := IOData2.Pt03.Data;
   	LastIOData[1].04 := IOData2.Pt04.Data;
   	LastIOData[1].05 := IOData2.Pt05.Data;
   	LastIOData[1].06 := IOData2.Pt06.Data;
   	LastIOData[1].07 := IOData2.Pt07.Data;
   	LastIOData[1].08 := IOData2.Pt08.Data;
   	LastIOData[1].09 := IOData2.Pt09.Data;
   	LastIOData[1].10 := IOData2.Pt10.Data;
   	LastIOData[1].11 := IOData2.Pt11.Data;
   	LastIOData[1].12 := IOData2.Pt12.Data;
   	LastIOData[1].13 := IOData2.Pt13.Data;
   	LastIOData[1].14 := IOData2.Pt14.Data;
   	LastIOData[1].15 := IOData2.Pt15.Data;
   	LastIOData[2].00 := IOData3.Pt00.Data;
   	LastIOData[2].01 := IOData3.Pt01.Data;
   	LastIOData[2].02 := IOData3.Pt02.Data;
   	LastIOData[2].03 := IOData3.Pt03.Data;
   	LastIOData[2].04 := IOData3.Pt04.Data;
   	LastIOData[2].05 := IOData3.Pt05.Data;
   	LastIOData[2].06 := IOData3.Pt06.Data;
   	LastIOData[2].07 := IOData3.Pt07.Data;
   	LastIOData[2].08 := IOData3.Pt08.Data;
   	LastIOData[2].09 := IOData3.Pt09.Data;
   	LastIOData[2].10 := IOData3.Pt10.Data;
   	LastIOData[2].11 := IOData3.Pt11.Data;
   	LastIOData[2].12 := IOData3.Pt12.Data;
   	LastIOData[2].13 := IOData3.Pt13.Data;
   	LastIOData[2].14 := IOData3.Pt14.Data;
   	LastIOData[2].15 := IOData3.Pt15.Data;
   	LastIOData[3].00 := IOData4.Pt00.Data;
   	LastIOData[3].01 := IOData4.Pt01.Data;
   	LastIOData[3].02 := IOData4.Pt02.Data;
   	LastIOData[3].03 := IOData4.Pt03.Data;
   	LastIOData[3].04 := IOData4.Pt04.Data;
   	LastIOData[3].05 := IOData4.Pt05.Data;
   	LastIOData[3].06 := IOData4.Pt06.Data;
   	LastIOData[3].07 := IOData4.Pt07.Data;
   	LastIOData[3].08 := IOData4.Pt08.Data;
   	LastIOData[3].09 := IOData4.Pt09.Data;
   	LastIOData[3].10 := IOData4.Pt10.Data;
   	LastIOData[3].11 := IOData4.Pt11.Data;
   	LastIOData[3].12 := IOData4.Pt12.Data;
   	LastIOData[3].13 := IOData4.Pt13.Data;
   	LastIOData[3].14 := IOData4.Pt14.Data;
   	LastIOData[3].15 := IOData4.Pt15.Data;
   	LastIOData[4].00 := IOData5.Pt00.Data;
   	LastIOData[4].01 := IOData5.Pt01.Data;
   	LastIOData[4].02 := IOData5.Pt02.Data;
   	LastIOData[4].03 := IOData5.Pt03.Data;
   	LastIOData[4].04 := IOData5.Pt04.Data;
   	LastIOData[4].05 := IOData5.Pt05.Data;
   	LastIOData[4].06 := IOData5.Pt06.Data;
   	LastIOData[4].07 := IOData5.Pt07.Data;
   	LastIOData[4].08 := IOData5.Pt08.Data;
   	LastIOData[4].09 := IOData5.Pt09.Data;
   	LastIOData[4].10 := IOData5.Pt10.Data;
   	LastIOData[4].11 := IOData5.Pt11.Data;
   	LastIOData[4].12 := IOData5.Pt12.Data;
   	LastIOData[4].13 := IOData5.Pt13.Data;
   	LastIOData[4].14 := IOData5.Pt14.Data;
   	LastIOData[4].15 := IOData5.Pt15.Data;
   	LastIOData[5].00 := IOData6.Pt00.Data;
   	LastIOData[5].01 := IOData6.Pt01.Data;
   	LastIOData[5].02 := IOData6.Pt02.Data;
   	LastIOData[5].03 := IOData6.Pt03.Data;
   	LastIOData[5].04 := IOData6.Pt04.Data;
   	LastIOData[5].05 := IOData6.Pt05.Data;
   	LastIOData[5].06 := IOData6.Pt06.Data;
   	LastIOData[5].07 := IOData6.Pt07.Data;
   	LastIOData[5].08 := IOData6.Pt08.Data;
   	LastIOData[5].09 := IOData6.Pt09.Data;
   	LastIOData[5].10 := IOData6.Pt10.Data;
   	LastIOData[5].11 := IOData6.Pt11.Data;
   	LastIOData[5].12 := IOData6.Pt12.Data;
   	LastIOData[5].13 := IOData6.Pt13.Data;
   	LastIOData[5].14 := IOData6.Pt14.Data;
   	LastIOData[5].15 := IOData6.Pt15.Data;
   	LastIOData[6].00 := IOData7.Pt00.Data;
   	LastIOData[6].01 := IOData7.Pt01.Data;
   	LastIOData[6].02 := IOData7.Pt02.Data;
   	LastIOData[6].03 := IOData7.Pt03.Data;
   	LastIOData[6].04 := IOData7.Pt04.Data;
   	LastIOData[6].05 := IOData7.Pt05.Data;
   	LastIOData[6].06 := IOData7.Pt06.Data;
   	LastIOData[6].07 := IOData7.Pt07.Data;
   	LastIOData[6].08 := IOData7.Pt08.Data;
   	LastIOData[6].09 := IOData7.Pt09.Data;
   	LastIOData[6].10 := IOData7.Pt10.Data;
   	LastIOData[6].11 := IOData7.Pt11.Data;
   	LastIOData[6].12 := IOData7.Pt12.Data;
   	LastIOData[6].13 := IOData7.Pt13.Data;
   	LastIOData[6].14 := IOData7.Pt14.Data;
   	LastIOData[6].15 := IOData7.Pt15.Data;
   	LastIOData[7].00 := IOData8.Pt00.Data;
   	LastIOData[7].01 := IOData8.Pt01.Data;
   	LastIOData[7].02 := IOData8.Pt02.Data;
   	LastIOData[7].03 := IOData8.Pt03.Data;
   	LastIOData[7].04 := IOData8.Pt04.Data;
   	LastIOData[7].05 := IOData8.Pt05.Data;
   	LastIOData[7].06 := IOData8.Pt06.Data;
   	LastIOData[7].07 := IOData8.Pt07.Data;
   	LastIOData[7].08 := IOData8.Pt08.Data;
   	LastIOData[7].09 := IOData8.Pt09.Data;
   	LastIOData[7].10 := IOData8.Pt10.Data;
   	LastIOData[7].11 := IOData8.Pt11.Data;
   	LastIOData[7].12 := IOData8.Pt12.Data;
   	LastIOData[7].13 := IOData8.Pt13.Data;
   	LastIOData[7].14 := IOData8.Pt14.Data;
   	LastIOData[7].15 := IOData8.Pt15.Data;
   else
   	CurrData[0].00 := IOData1.Pt00.Data;
   	CurrData[0].01 := IOData1.Pt01.Data;
   	CurrData[0].02 := IOData1.Pt02.Data;
   	CurrData[0].03 := IOData1.Pt03.Data;
   	CurrData[0].04 := IOData1.Pt04.Data;
   	CurrData[0].05 := IOData1.Pt05.Data;
   	CurrData[0].06 := IOData1.Pt06.Data;
   	CurrData[0].07 := IOData1.Pt07.Data;
   	CurrData[0].08 := IOData1.Pt08.Data;
   	CurrData[0].09 := IOData1.Pt09.Data;
   	CurrData[0].10 := IOData1.Pt10.Data;
   	CurrData[0].11 := IOData1.Pt11.Data;
   	CurrData[0].12 := IOData1.Pt12.Data;
   	CurrData[0].13 := IOData1.Pt13.Data;
   	CurrData[0].14 := IOData1.Pt14.Data;
   	CurrData[0].15 := IOData1.Pt15.Data;
   	CurrData[1].00 := IOData2.Pt00.Data;
   	CurrData[1].01 := IOData2.Pt01.Data;
   	CurrData[1].02 := IOData2.Pt02.Data;
   	CurrData[1].03 := IOData2.Pt03.Data;
   	CurrData[1].04 := IOData2.Pt04.Data;
   	CurrData[1].05 := IOData2.Pt05.Data;
   	CurrData[1].06 := IOData2.Pt06.Data;
   	CurrData[1].07 := IOData2.Pt07.Data;
   	CurrData[1].08 := IOData2.Pt08.Data;
   	CurrData[1].09 := IOData2.Pt09.Data;
   	CurrData[1].10 := IOData2.Pt10.Data;
   	CurrData[1].11 := IOData2.Pt11.Data;
   	CurrData[1].12 := IOData2.Pt12.Data;
   	CurrData[1].13 := IOData2.Pt13.Data;
   	CurrData[1].14 := IOData2.Pt14.Data;
   	CurrData[1].15 := IOData2.Pt15.Data;
   	CurrData[2].00 := IOData3.Pt00.Data;
   	CurrData[2].01 := IOData3.Pt01.Data;
   	CurrData[2].02 := IOData3.Pt02.Data;
   	CurrData[2].03 := IOData3.Pt03.Data;
   	CurrData[2].04 := IOData3.Pt04.Data;
   	CurrData[2].05 := IOData3.Pt05.Data;
   	CurrData[2].06 := IOData3.Pt06.Data;
   	CurrData[2].07 := IOData3.Pt07.Data;
   	CurrData[2].08 := IOData3.Pt08.Data;
   	CurrData[2].09 := IOData3.Pt09.Data;
   	CurrData[2].10 := IOData3.Pt10.Data;
   	CurrData[2].11 := IOData3.Pt11.Data;
   	CurrData[2].12 := IOData3.Pt12.Data;
   	CurrData[2].13 := IOData3.Pt13.Data;
   	CurrData[2].14 := IOData3.Pt14.Data;
   	CurrData[2].15 := IOData3.Pt15.Data;
   	CurrData[3].00 := IOData4.Pt00.Data;
   	CurrData[3].01 := IOData4.Pt01.Data;
   	CurrData[3].02 := IOData4.Pt02.Data;
   	CurrData[3].03 := IOData4.Pt03.Data;
   	CurrData[3].04 := IOData4.Pt04.Data;
   	CurrData[3].05 := IOData4.Pt05.Data;
   	CurrData[3].06 := IOData4.Pt06.Data;
   	CurrData[3].07 := IOData4.Pt07.Data;
   	CurrData[3].08 := IOData4.Pt08.Data;
   	CurrData[3].09 := IOData4.Pt09.Data;
   	CurrData[3].10 := IOData4.Pt10.Data;
   	CurrData[3].11 := IOData4.Pt11.Data;
   	CurrData[3].12 := IOData4.Pt12.Data;
   	CurrData[3].13 := IOData4.Pt13.Data;
   	CurrData[3].14 := IOData4.Pt14.Data;
   	CurrData[3].15 := IOData4.Pt15.Data;
   	CurrData[4].00 := IOData5.Pt00.Data;
   	CurrData[4].01 := IOData5.Pt01.Data;
   	CurrData[4].02 := IOData5.Pt02.Data;
   	CurrData[4].03 := IOData5.Pt03.Data;
   	CurrData[4].04 := IOData5.Pt04.Data;
   	CurrData[4].05 := IOData5.Pt05.Data;
   	CurrData[4].06 := IOData5.Pt06.Data;
   	CurrData[4].07 := IOData5.Pt07.Data;
   	CurrData[4].08 := IOData5.Pt08.Data;
   	CurrData[4].09 := IOData5.Pt09.Data;
   	CurrData[4].10 := IOData5.Pt10.Data;
   	CurrData[4].11 := IOData5.Pt11.Data;
   	CurrData[4].12 := IOData5.Pt12.Data;
   	CurrData[4].13 := IOData5.Pt13.Data;
   	CurrData[4].14 := IOData5.Pt14.Data;
   	CurrData[4].15 := IOData5.Pt15.Data;
   	CurrData[5].00 := IOData6.Pt00.Data;
   	CurrData[5].01 := IOData6.Pt01.Data;
   	CurrData[5].02 := IOData6.Pt02.Data;
   	CurrData[5].03 := IOData6.Pt03.Data;
   	CurrData[5].04 := IOData6.Pt04.Data;
   	CurrData[5].05 := IOData6.Pt05.Data;
   	CurrData[5].06 := IOData6.Pt06.Data;
   	CurrData[5].07 := IOData6.Pt07.Data;
   	CurrData[5].08 := IOData6.Pt08.Data;
   	CurrData[5].09 := IOData6.Pt09.Data;
   	CurrData[5].10 := IOData6.Pt10.Data;
   	CurrData[5].11 := IOData6.Pt11.Data;
   	CurrData[5].12 := IOData6.Pt12.Data;
   	CurrData[5].13 := IOData6.Pt13.Data;
   	CurrData[5].14 := IOData6.Pt14.Data;
   	CurrData[5].15 := IOData6.Pt15.Data;
   	CurrData[6].00 := IOData7.Pt00.Data;
   	CurrData[6].01 := IOData7.Pt01.Data;
   	CurrData[6].02 := IOData7.Pt02.Data;
   	CurrData[6].03 := IOData7.Pt03.Data;
   	CurrData[6].04 := IOData7.Pt04.Data;
   	CurrData[6].05 := IOData7.Pt05.Data;
   	CurrData[6].06 := IOData7.Pt06.Data;
   	CurrData[6].07 := IOData7.Pt07.Data;
   	CurrData[6].08 := IOData7.Pt08.Data;
   	CurrData[6].09 := IOData7.Pt09.Data;
   	CurrData[6].10 := IOData7.Pt10.Data;
   	CurrData[6].11 := IOData7.Pt11.Data;
   	CurrData[6].12 := IOData7.Pt12.Data;
   	CurrData[6].13 := IOData7.Pt13.Data;
   	CurrData[6].14 := IOData7.Pt14.Data;
   	CurrData[6].15 := IOData7.Pt15.Data;
   	CurrData[7].00 := IOData8.Pt00.Data;
   	CurrData[7].01 := IOData8.Pt01.Data;
   	CurrData[7].02 := IOData8.Pt02.Data;
   	CurrData[7].03 := IOData8.Pt03.Data;
   	CurrData[7].04 := IOData8.Pt04.Data;
   	CurrData[7].05 := IOData8.Pt05.Data;
   	CurrData[7].06 := IOData8.Pt06.Data;
   	CurrData[7].07 := IOData8.Pt07.Data;
   	CurrData[7].08 := IOData8.Pt08.Data;
   	CurrData[7].09 := IOData8.Pt09.Data;
   	CurrData[7].10 := IOData8.Pt10.Data;
   	CurrData[7].11 := IOData8.Pt11.Data;
   	CurrData[7].12 := IOData8.Pt12.Data;
   	CurrData[7].13 := IOData8.Pt13.Data;
   	CurrData[7].14 := IOData8.Pt14.Data;
   	CurrData[7].15 := IOData8.Pt15.Data;
   
   	for index := 0 to 7 do
   		for bindex := 0 to 15 do
   			if (CurrData[index] AND 2**bindex)=0 AND (LastIOData[index] AND 2**bindex)<>0 then
   				CounterArray[index*8+bindex] := CounterArray[index*8+bindex]+1;
   			end_if;
   		end_for;
   	end_for;
   
   	CPS(CurrData[0],LastIOData[0],8);
   end_if;
   
   for index := 0 to 7 do
   	for bindex := 0 to 15 do
   		if (ResetArray[index] AND 2**bindex)>0 then
   			CounterArray[index*16+bindex] := 0;
   		end_if;
   	end_for;
   end_for;
END_ROUTINE
END_ADD_ON_INSTRUCTION

ADD_ON_INSTRUCTION AOI_KeyenceBarcode   (* revision 1.0 *)
VAR_IN_OUT
   Input : udt_KeyenceScannerInputs; {required}
   Output : udt_KeyenceScannerOutputs; {required}
END_VAR
VAR_INPUT
   Trigger : BOOL; {access Read Only}
   HandshakeEnabled : BOOL; {access Read Only}
END_VAR
VAR_OUTPUT
   ReadSuccess : BOOL;
END_VAR
VAR_IN_OUT
   BarcodeValue : STR_Barcode; {required}
END_VAR
VAR_INPUT
   RetrieveResultData : BOOL; {access Read Only}
END_VAR
VAR
   Ready : BOOL; {access None}
END_VAR

ROUTINE Logic   (* ladder *)
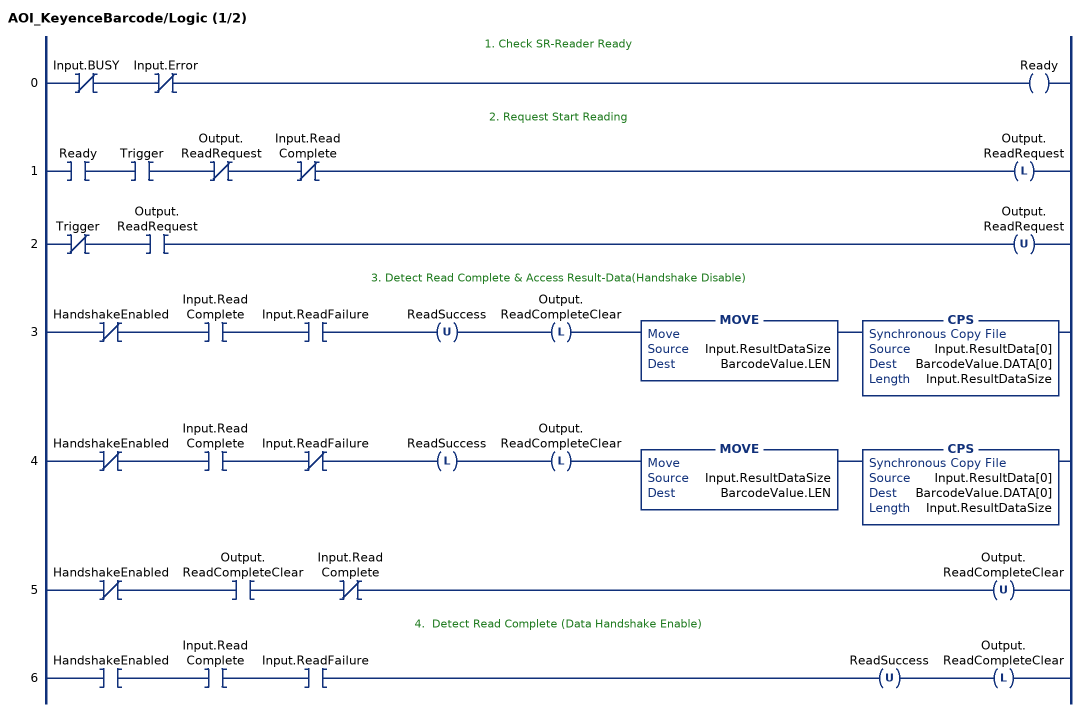
   // 1. Check SR-Reader Ready
   0: XIO(Input.BUSY)XIO(Input.Error)OTE(Ready);
   // 2. Request Start Reading
   1: XIC(Ready)XIC(Trigger)XIO(Output.ReadRequest)XIO(Input.ReadComplete)OTL(Output.ReadRequest);
   2: XIO(Trigger)XIC(Output.ReadRequest)OTU(Output.ReadRequest);
   // 3. Detect Read Complete & Access Result-Data(Handshake Disable)
   3: XIO(HandshakeEnabled)XIC(Input.ReadComplete)XIC(Input.ReadFailure)OTU(ReadSuccess)OTL(Output.ReadCompleteClear)MOVE(Input.ResultDataSize,BarcodeValue.LEN)CPS(Input.ResultData[0],BarcodeValue.DATA[0],Input.ResultDataSize);
   4: XIO(HandshakeEnabled)XIC(Input.ReadComplete)XIO(Input.ReadFailure)OTL(ReadSuccess)OTL(Output.ReadCompleteClear)MOVE(Input.ResultDataSize,BarcodeValue.LEN)CPS(Input.ResultData[0],BarcodeValue.DATA[0],Input.ResultDataSize);
   5: XIO(HandshakeEnabled)XIC(Output.ReadCompleteClear)XIO(Input.ReadComplete)OTU(Output.ReadCompleteClear);
   // 4.  Detect Read Complete (Data Handshake Enable)
   6: XIC(HandshakeEnabled)XIC(Input.ReadComplete)XIC(Input.ReadFailure)OTU(ReadSuccess)OTL(Output.ReadCompleteClear);
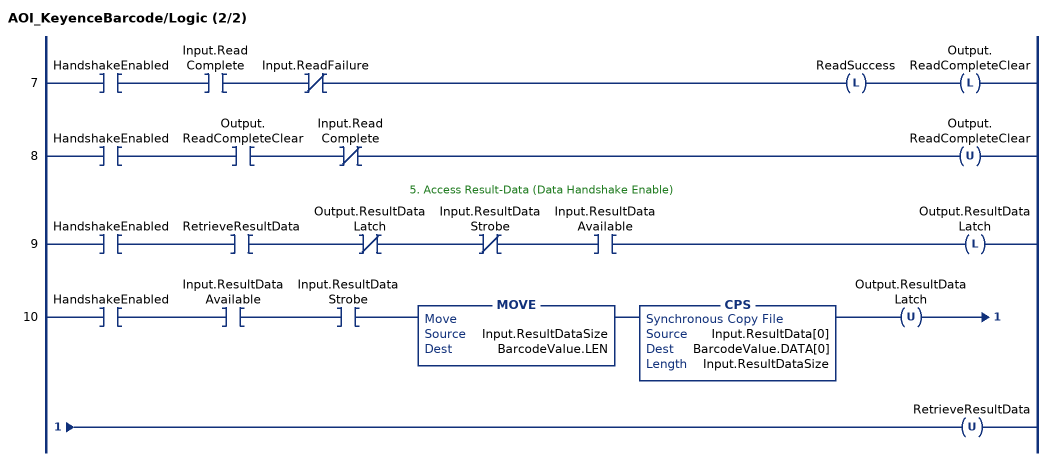
   7: XIC(HandshakeEnabled)XIC(Input.ReadComplete)XIO(Input.ReadFailure)OTL(ReadSuccess)OTL(Output.ReadCompleteClear);
   8: XIC(HandshakeEnabled)XIC(Output.ReadCompleteClear)XIO(Input.ReadComplete)OTU(Output.ReadCompleteClear);
   // 5. Access Result-Data (Data Handshake Enable)
   9: XIC(HandshakeEnabled)XIC(RetrieveResultData)XIO(Output.ResultDataLatch)XIO(Input.ResultDataStrobe)XIC(Input.ResultDataAvailable)OTL(Output.ResultDataLatch);
   10: XIC(HandshakeEnabled)XIC(Input.ResultDataAvailable)XIC(Input.ResultDataStrobe)MOVE(Input.ResultDataSize,BarcodeValue.LEN)CPS(Input.ResultData[0],BarcodeValue.DATA[0],Input.ResultDataSize)OTU(Output.ResultDataLatch)OTU(RetrieveResultData);
END_ROUTINE
END_ADD_ON_INSTRUCTION

ADD_ON_INSTRUCTION AOI_PLC   (* revision 1.0 *)
VAR_OUTPUT
   AlwaysOn : BOOL; {visible}
   AlwaysOff : BOOL; {visible}
   FlasherSlow : BOOL; {visible}
   FlasherMedium : BOOL; {visible}
   FlasherFast : BOOL; {visible}
   FirstScan : BOOL; {access Read Only, visible}
END_VAR
VAR_INPUT
   xxxxxx_FLASHER_SETTINGS_xxxxxx : BOOL; {visible}
   SlowFlashTime : DINT; {visible}
   MediumFlashTime : DINT; {visible}
   FastFlashTime : DINT; {visible}
   UseRemoteFlashers : BOOL; {visible}
   FlasherSlowInput : BOOL; {visible}
   FlasherMediumInput : BOOL; {visible}
   FlasherFastInput : BOOL; {visible}
   xxxxxx_PLC_DATE_AND_TIME_xxxxxx : BOOL; {visible}
END_VAR
VAR_OUTPUT
   Year : INT; {access Read Only, visible}
   Day : INT; {access Read Only, visible}
   Month : INT; {access Read Only, visible}
   Hour : INT; {access Read Only, visible}
   Minute : INT; {access Read Only, visible}
   Second : INT; {access Read Only, visible}
   MicroSecond : DINT; {access Read Only, visible}
END_VAR
VAR_INPUT
   DOY : INT; {access Read Only, visible}
END_VAR
VAR_IN_OUT
   DateString : String20; {required}
   TimeString : String20; {required}
   DateTimeString : String20; {required}
END_VAR
VAR_INPUT
   xxxxxx_PLC_EDIT_HISTORY_xxxxxx : BOOL; {visible}
END_VAR
VAR_IN_OUT
   LastPLCEdit : String20; {required}
   LastPLCEditHistory : String20[20]; {required}
END_VAR
VAR_OUTPUT
   TimeSyncStrobe : BOOL; {access Read Only}
END_VAR
VAR_INPUT
   SetTimePB : BOOL;
   SetYear : INT;
   SetMonth : INT;
   SetDay : INT;
   SetHour : INT;
   SetMinute : INT;
   SetSecond : INT;
END_VAR
VAR
   SlowTON : TIMER; {access None}
   Medium_TON : TIMER; {access None}
   Fast_TON : TIMER; {access None}
   SlowLimit : DINT; {access None}
   MediumLimit : DINT; {access None}
   FastLimit : DINT; {access None}
   YearString : String20; {access None}
   TimeStringTemp : String20; {access None}
   Space : String20; {access None}
   Slash : String20; {access None}
   SecondString : String20; {access None}
   MonthString : String20; {access None}
   MinuteString : String20; {access None}
   HourString : String20; {access None}
   DayString : String20; {access None}
   DateTime : DINT[7]; {access None}
   DateTimeStringTemp : String20; {access None}
   DateStringTemp : String20; {access None}
   Colon : String20; {access None}
   AUDIT_VALUE_DINT : DINT[2]; {access None}
   PLC_EditHistory_TON : TIMER := (PRE := 2000, ACC := 511); {access None}
   PLC_EditHistory_ONS : BOOL; {access None}
   AUDIT_VALUE_LAST : DINT[2]; {access None}
   LastPLCEditHistoryTemp : String20[20]; {access None}
   HourHistory : SINT; {access None}
   TimeSyncTMR : TIMER := (PRE := 1000); {access None}
   DayArray : INT[13] := ([2] := 31, [3] := 59, [4] := 90, [5] := 120, [6] := 151, [7] := 181, [8] := 212, [9] := 243, [10] := 273, [11] := 304, [12] := 334); {access None}
   ZeroString : String20 := '0'; {access None}
END_VAR

ROUTINE Logic   (* ladder *)
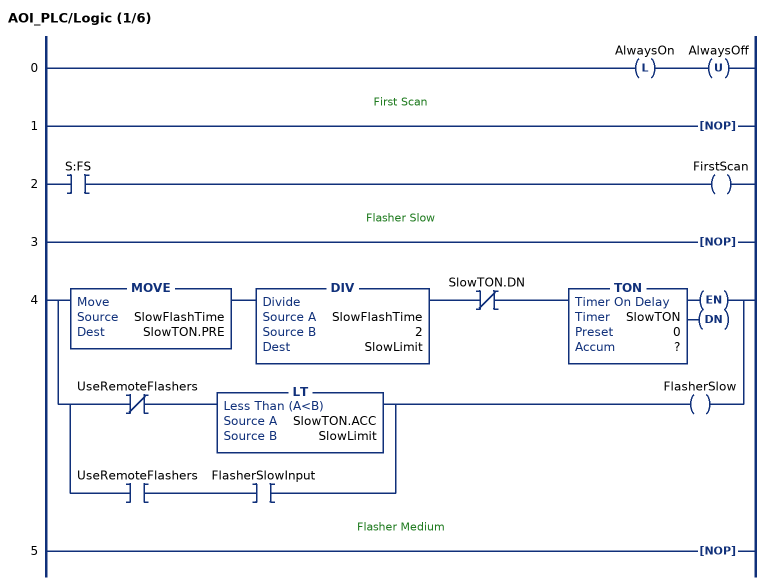
   0: OTL(AlwaysOn)OTU(AlwaysOff);
   // First Scan
   1: NOP();
   2: XIC(S:FS)OTE(FirstScan);
   // Flasher Slow
   3: NOP();
   4: [MOVE(SlowFlashTime,SlowTON.PRE) DIV(SlowFlashTime,2,SlowLimit) XIO(SlowTON.DN) TON(SlowTON,?,?) ,[XIO(UseRemoteFlashers) LT(SlowTON.ACC,SlowLimit) ,XIC(UseRemoteFlashers) XIC(FlasherSlowInput) ] OTE(FlasherSlow) ];
   // Flasher Medium
   5: NOP();
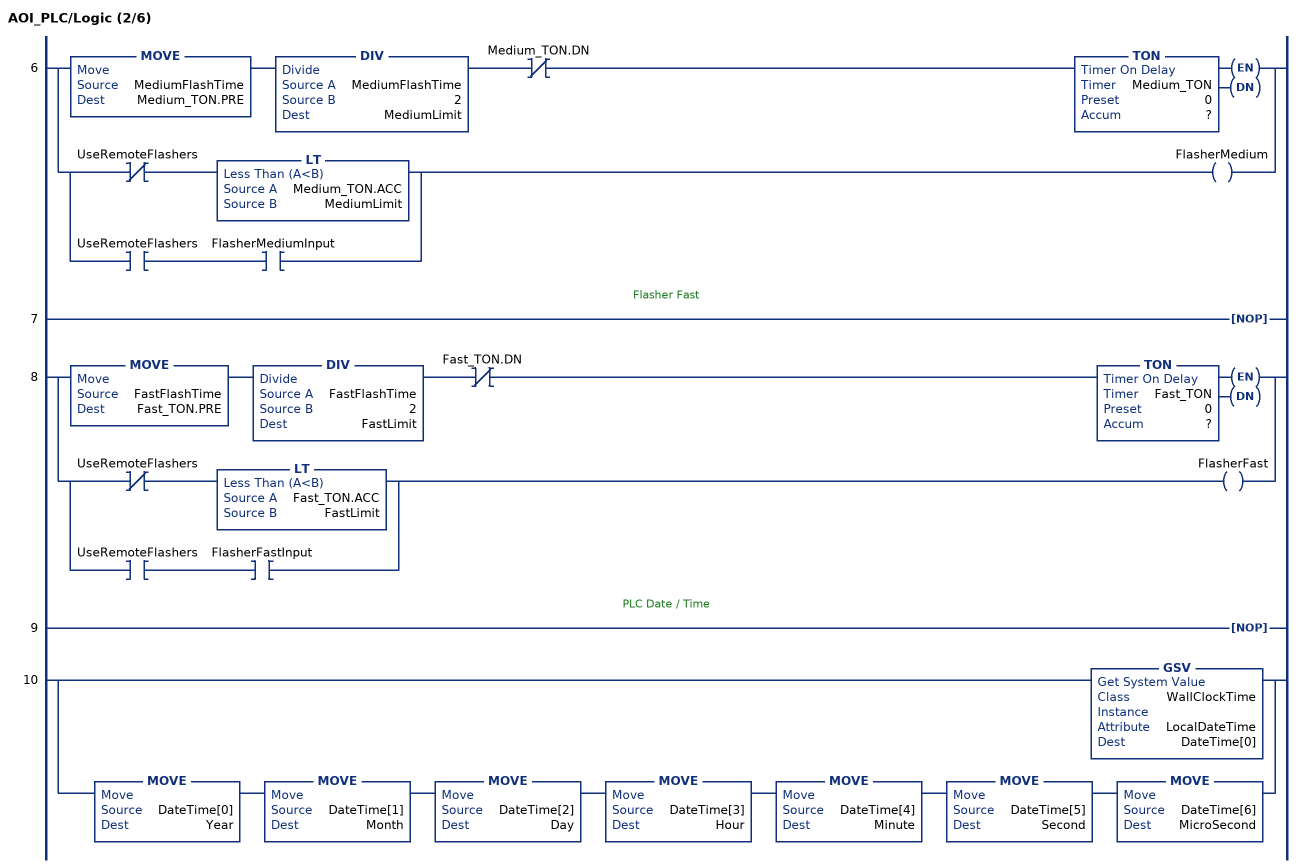
   6: [MOVE(MediumFlashTime,Medium_TON.PRE) DIV(MediumFlashTime,2,MediumLimit) XIO(Medium_TON.DN) TON(Medium_TON,?,?) ,[XIO(UseRemoteFlashers) LT(Medium_TON.ACC,MediumLimit) ,XIC(UseRemoteFlashers) XIC(FlasherMediumInput) ] OTE(FlasherMedium) ];
   // Flasher Fast
   7: NOP();
   8: [MOVE(FastFlashTime,Fast_TON.PRE) DIV(FastFlashTime,2,FastLimit) XIO(Fast_TON.DN) TON(Fast_TON,?,?) ,[XIO(UseRemoteFlashers) LT(Fast_TON.ACC,FastLimit) ,XIC(UseRemoteFlashers) XIC(FlasherFastInput) ] OTE(FlasherFast) ];
   // PLC Date / Time
   9: NOP();
   10: [GSV(WallClockTime,,LocalDateTime,DateTime[0]) ,MOVE(DateTime[0],Year) MOVE(DateTime[1],Month) MOVE(DateTime[2],Day) MOVE(DateTime[3],Hour) MOVE(DateTime[4],Minute) MOVE(DateTime[5],Second) MOVE(DateTime[6],MicroSecond) ];
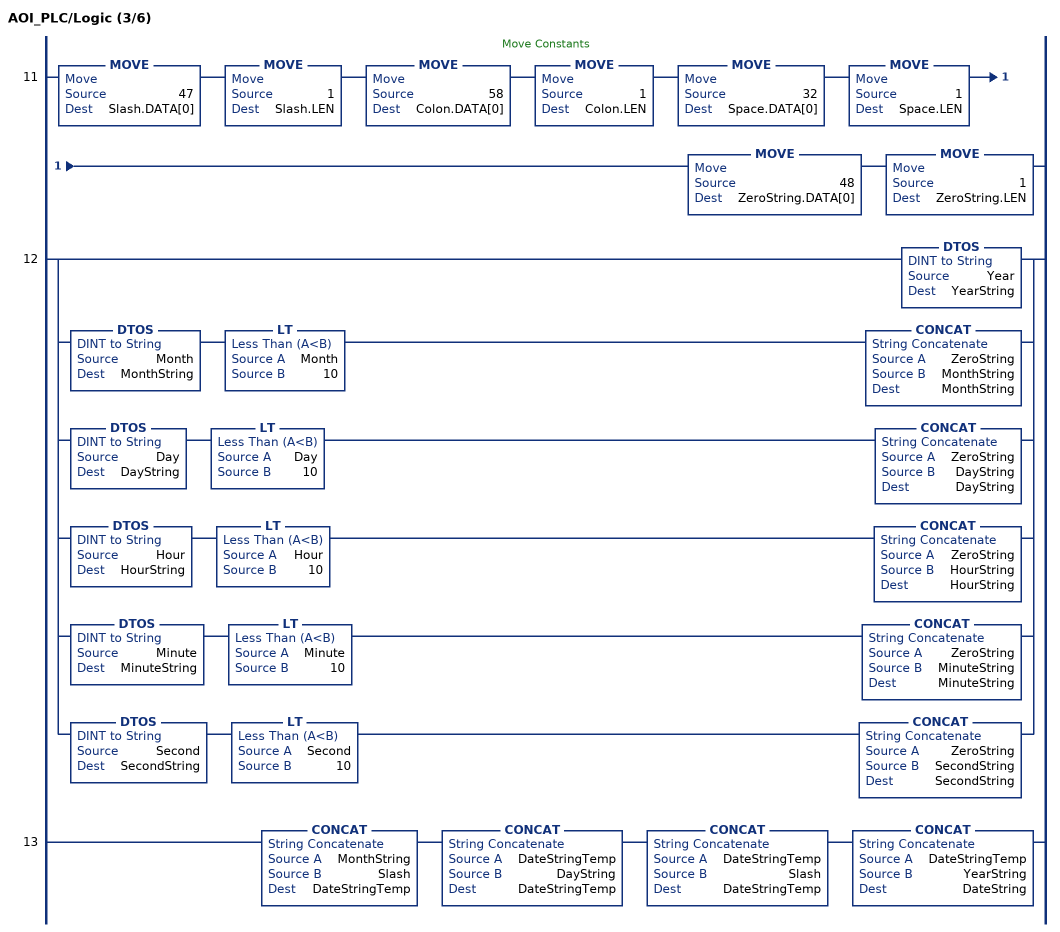
   // Move Constants
   11: MOVE(47,Slash.DATA[0])MOVE(1,Slash.LEN)MOVE(58,Colon.DATA[0])MOVE(1,Colon.LEN)MOVE(32,Space.DATA[0])MOVE(1,Space.LEN)MOVE(48,ZeroString.DATA[0])MOVE(1,ZeroString.LEN);
   12: [DTOS(Year,YearString) ,DTOS(Month,MonthString) LT(Month,10) CONCAT(ZeroString,MonthString,MonthString) ,DTOS(Day,DayString) LT(Day,10) CONCAT(ZeroString,DayString,DayString) ,DTOS(Hour,HourString) LT(Hour,10) CONCAT(ZeroString,HourString,HourString) ,DTOS(Minute,MinuteString) LT(Minute,10) CONCAT(ZeroString,MinuteString,MinuteString) ,DTOS(Second,SecondString) LT(Second,10) CONCAT(ZeroString,SecondString,SecondString) ];
   13: CONCAT(MonthString,Slash,DateStringTemp)CONCAT(DateStringTemp,DayString,DateStringTemp)CONCAT(DateStringTemp,Slash,DateStringTemp)CONCAT(DateStringTemp,YearString,DateString);
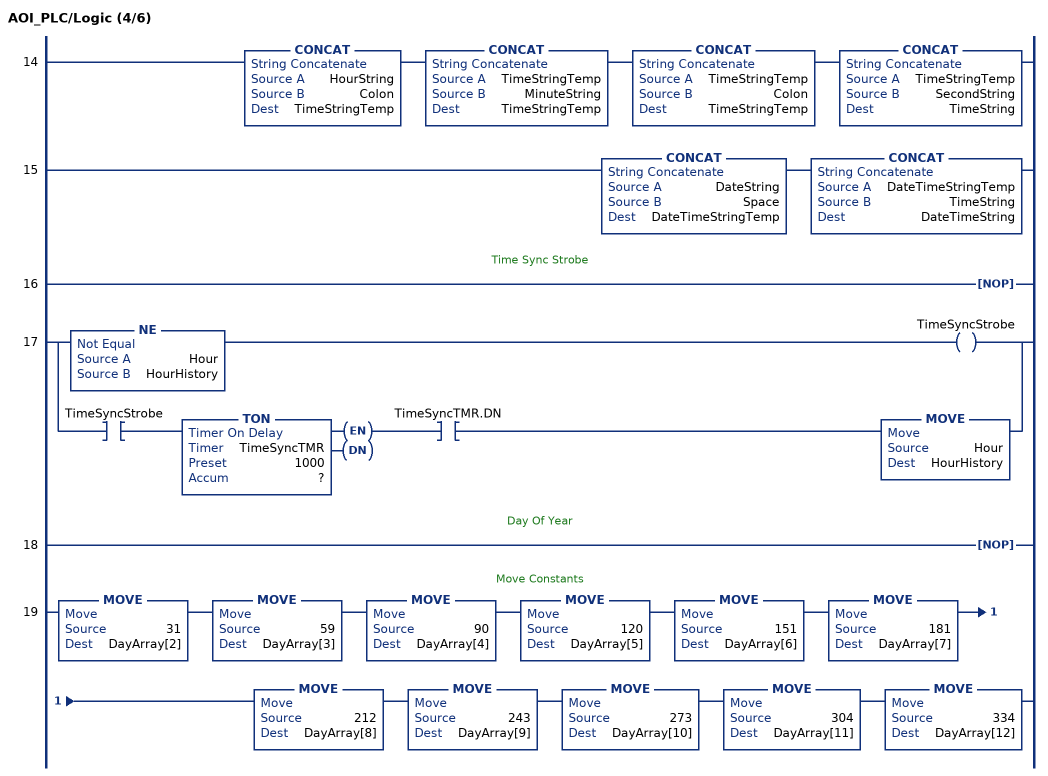
   14: CONCAT(HourString,Colon,TimeStringTemp)CONCAT(TimeStringTemp,MinuteString,TimeStringTemp)CONCAT(TimeStringTemp,Colon,TimeStringTemp)CONCAT(TimeStringTemp,SecondString,TimeString);
   15: CONCAT(DateString,Space,DateTimeStringTemp)CONCAT(DateTimeStringTemp,TimeString,DateTimeString);
   // Time Sync Strobe
   16: NOP();
   17: [NE(Hour,HourHistory) OTE(TimeSyncStrobe) ,XIC(TimeSyncStrobe) TON(TimeSyncTMR,?,?) XIC(TimeSyncTMR.DN) MOVE(Hour,HourHistory) ];
   // Day Of Year
   18: NOP();
   // Move Constants
   19: MOVE(31,DayArray[2])MOVE(59,DayArray[3])MOVE(90,DayArray[4])MOVE(120,DayArray[5])MOVE(151,DayArray[6])MOVE(181,DayArray[7])MOVE(212,DayArray[8])MOVE(243,DayArray[9])MOVE(273,DayArray[10])MOVE(304,DayArray[11])MOVE(334,DayArray[12]);
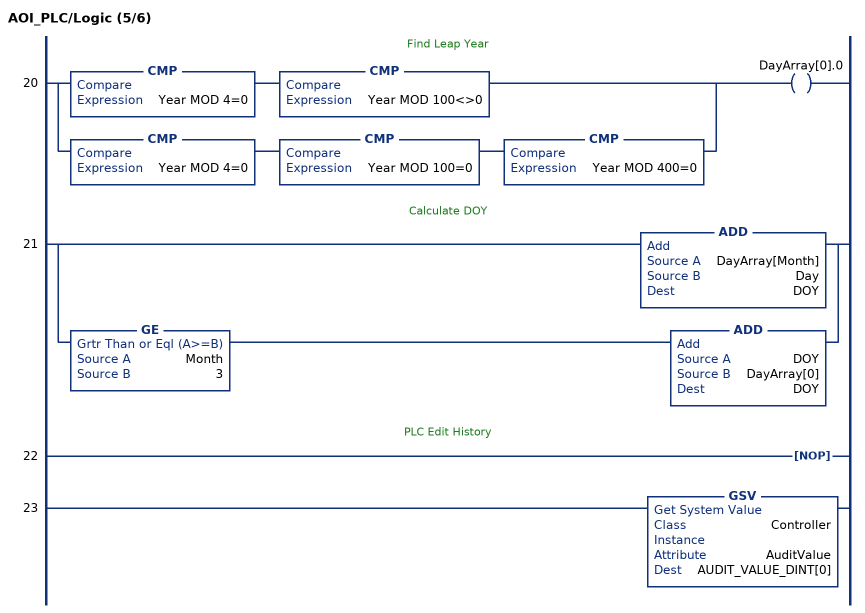
   // Find Leap Year
   20: [CMP(Year MOD 4=0) CMP(Year MOD 100<>0) ,CMP(Year MOD 4=0) CMP(Year MOD 100=0) CMP(Year MOD 400=0) ]OTE(DayArray[0].0);
   // Calculate DOY
   21: [ADD(DayArray[Month],Day,DOY) ,GE(Month,3) ADD(DOY,DayArray[0],DOY) ];
   // PLC Edit History
   22: NOP();
   23: GSV(Controller,,AuditValue,AUDIT_VALUE_DINT[0]);
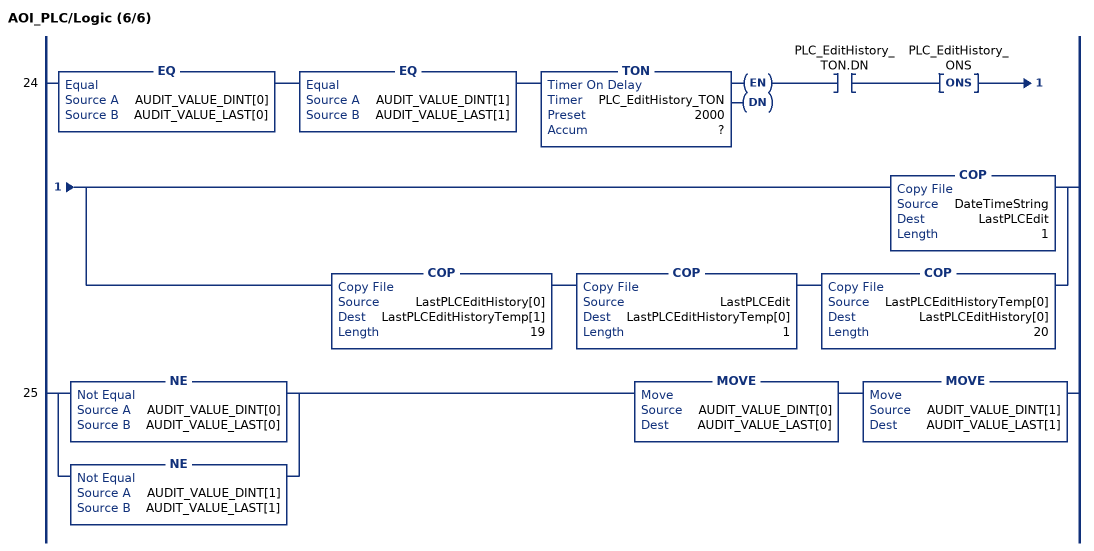
   24: EQ(AUDIT_VALUE_DINT[0],AUDIT_VALUE_LAST[0])EQ(AUDIT_VALUE_DINT[1],AUDIT_VALUE_LAST[1])TON(PLC_EditHistory_TON,?,?)XIC(PLC_EditHistory_TON.DN)ONS(PLC_EditHistory_ONS)[COP(DateTimeString,LastPLCEdit,1) ,COP(LastPLCEditHistory[0],LastPLCEditHistoryTemp[1],19) COP(LastPLCEdit,LastPLCEditHistoryTemp[0],1) COP(LastPLCEditHistoryTemp[0],LastPLCEditHistory[0],20) ];
   25: [NE(AUDIT_VALUE_DINT[0],AUDIT_VALUE_LAST[0]) ,NE(AUDIT_VALUE_DINT[1],AUDIT_VALUE_LAST[1]) ]MOVE(AUDIT_VALUE_DINT[0],AUDIT_VALUE_LAST[0])MOVE(AUDIT_VALUE_DINT[1],AUDIT_VALUE_LAST[1]);
END_ROUTINE
END_ADD_ON_INSTRUCTION
